ACTION ACT_LoopRead:
loopreadConditionTON(IN:=NOT setBusy AND NOT readBusy AND NOT gTBPStopLoopRead,PT:=T#1S);
IF loopreadConditionTON.Q THEN
	loopReadExcute:=TRUE;
END_IF
CASE loopReadStep OF
	0:
		IF loopReadExcute THEN
			loopReadExcute:=FALSE;
			loopReadStep:=10;
			readBusy:=TRUE;
			t1(IN:=FALSE);
			t2(IN:=FALSE);
		END_IF
	10:
		readDone:=FALSE;
		Read_State_1();
		t1(IN:=FALSE);
		loopReadStep:=loopReadStep+10;
	20:
		IF readDone THEN
			readDone:=FALSE;
			loopReadStep:=loopReadStep+10;
			t1(IN:=FALSE);
			RETURN;
		END_IF
		t1(IN:=TRUE,PT:=T#200MS);
		IF t1.Q THEN
			serialTimeOut:=TRUE;
			t1(IN:=FALSE);
			loopReadStep:=6000;
			t1(IN:=FALSE);
			RETURN;
		END_IF
	30:
		t2(IN:=TRUE,PT:=timeToNext);
		IF t2.Q THEN
			loopReadStep:=loopReadStep+10;
			t1(IN:=FALSE);
			t2(IN:=FALSE);
			RETURN;
		END_IF
	40:
		readDone:=FALSE;
		Read_State_2();
		t1(IN:=FALSE);
		loopReadStep:=loopReadStep+10;
	50:
		IF readDone THEN
			readDone:=FALSE;
			loopReadStep:=loopReadStep+10;
			t1(IN:=FALSE);
			RETURN;
		END_IF
		t1(IN:=TRUE,PT:=T#200MS);
		IF t1.Q THEN
			serialTimeOut:=TRUE;
			t1(IN:=FALSE);
			loopReadStep:=6000;
			t1(IN:=FALSE);
			RETURN;
		END_IF
	60:
		t2(IN:=TRUE,PT:=timeToNext);
		IF t2.Q THEN
			loopReadStep:=loopReadStep+10;
			t1(IN:=FALSE);
			t2(IN:=FALSE);
			RETURN;
		END_IF
	70:
		readDone:=FALSE;
		Read_State_3();
		t1(IN:=FALSE);
		loopReadStep:=loopReadStep+10;
	80:
		IF readDone THEN
			readDone:=FALSE;
			loopReadStep:=loopReadStep+10;
			t1(IN:=FALSE);
			RETURN;
		END_IF
		t1(IN:=TRUE,PT:=T#200MS);
		IF t1.Q THEN
			serialTimeOut:=TRUE;
			t1(IN:=FALSE);
			loopReadStep:=6000;
			t1(IN:=FALSE);
			RETURN;
		END_IF
	90:
		t2(IN:=TRUE,PT:=timeToNext);
		IF t2.Q THEN
			loopReadStep:=loopReadStep+10;
			t1(IN:=FALSE);
			t2(IN:=FALSE);
			RETURN;
		END_IF
	100:
		readDone:=FALSE;
		Read_State_4();
		t1(IN:=FALSE);
		loopReadStep:=loopReadStep+10;
	110:
		IF readDone THEN
			readDone:=FALSE;
			// 低位
			atTagetSpeed:=arr_RcvDataByte[6].5;
			alarm:=arr_RcvDataByte[6].3 OR arr_RcvDataByte[6].2;
			remote:=arr_RcvDataByte[6].0;
			// 高位
			acc:=arr_RcvDataByte[7].7;
			brake:=arr_RcvDataByte[7].6;
			noRotation:=arr_RcvDataByte[7].5 (*OR NOT arr_RcvDataByte[7].1*);
			loopReadStep:=loopReadStep+10;
			t1(IN:=FALSE);
			RETURN;
		END_IF
		t1(IN:=TRUE,PT:=T#200MS);
		IF t1.Q THEN
			serialTimeOut:=TRUE;
			t1(IN:=FALSE);
			loopReadStep:=6000;
			t1(IN:=FALSE);
			RETURN;
		END_IF
	120:
		t2(IN:=TRUE,PT:=timeToNext);
		IF t2.Q THEN
			t1(IN:=FALSE);
			t2(IN:=FALSE);
			loopToReadRatationTimes:=loopToReadRatationTimes+1;
			IF loopToReadRatationTimes>2 THEN // 状态读取5次，转速更新一次
				loopReadStep:=200;// 读取转速
				loopToReadRatationTimes:=0;
			ELSE
				loopReadStep:=5000;
			END_IF
			RETURN;
		END_IF
	200:
		readDone:=FALSE;
		Read_Rotation_1();
		t1(IN:=FALSE);
		loopReadStep:=loopReadStep+10;
	210:
		IF readDone THEN
			readDone:=FALSE;
			loopReadStep:=loopReadStep+10;
			t1(IN:=FALSE);
			RETURN;
		END_IF
		t1(IN:=TRUE,PT:=T#200MS);
		IF t1.Q THEN
			serialTimeOut:=TRUE;
			t1(IN:=FALSE);
			loopReadStep:=6000;
			t1(IN:=FALSE);
			RETURN;
		END_IF
	220:
		t2(IN:=TRUE,PT:=timeToNext);
		IF t2.Q THEN
			loopReadStep:=loopReadStep+10;
			t1(IN:=FALSE);
			t2(IN:=FALSE);
			RETURN;
		END_IF
	230:
		readDone:=FALSE;
		Read_Rotation_2();
		t1(IN:=FALSE);
		loopReadStep:=loopReadStep+10;
	240:
		IF readDone THEN
			readDone:=FALSE;
			loopReadStep:=loopReadStep+10;
			t1(IN:=FALSE);
			RETURN;
		END_IF
		t1(IN:=TRUE,PT:=T#200MS);
		IF t1.Q THEN
			serialTimeOut:=TRUE;
			t1(IN:=FALSE);
			loopReadStep:=6000;
			t1(IN:=FALSE);
			RETURN;
		END_IF
	250:
		t2(IN:=TRUE,PT:=timeToNext);
		IF t2.Q THEN
			loopReadStep:=loopReadStep+10;
			t1(IN:=FALSE);
			t2(IN:=FALSE);
			RETURN;
		END_IF
	260:
		readDone:=FALSE;
		Read_Rotation_3();
		t1(IN:=FALSE);
		loopReadStep:=loopReadStep+10;
	270:
		IF readDone THEN
			readDone:=FALSE;
			loopReadStep:=loopReadStep+10;
			t1(IN:=FALSE);
			RETURN;
		END_IF
		t1(IN:=TRUE,PT:=T#200MS);
		IF t1.Q THEN
			serialTimeOut:=TRUE;
			t1(IN:=FALSE);
			loopReadStep:=6000;
			RETURN;
		END_IF
	280:
		t2(IN:=TRUE,PT:=timeToNext);
		IF t2.Q THEN
			loopReadStep:=loopReadStep+10;
			t1(IN:=FALSE);
			t2(IN:=FALSE);
			RETURN;
		END_IF
	290:
		readDone:=FALSE;
		Read_Rotation_4();
		t1(IN:=FALSE);
		loopReadStep:=loopReadStep+10;
	300:
		IF readDone THEN
			readDone:=FALSE;
			intTemp:=BYTE_TO_UDINT(arr_RcvDataByte[6])*256;// 读取转速进行转换 高位
			rotationSpeed:=(intTemp+BYTE_TO_UDINT(arr_RcvDataByte[7]));// 读取转速进行转换 低位   *60  HZ 
			loopReadStep:=loopReadStep+10;
			t1(IN:=FALSE);
			RETURN;
		END_IF
		t1(IN:=TRUE,PT:=T#200MS);
		IF t1.Q THEN
			serialTimeOut:=TRUE;
			t1(IN:=FALSE);
			loopReadStep:=6000;
			t1(IN:=FALSE);
			RETURN;
		END_IF
	310:
		t2(IN:=TRUE,PT:=timeToNext);
		IF t2.Q THEN
			loopReadStep:=loopReadStep+10;
			RETURN;
		END_IF
	320:
		loopReadStep:=400;
		
	400:
		readDone:=FALSE;
		Read_TMS_1();
		t1(IN:=FALSE);
		loopReadStep:=loopReadStep+10;
	410:
		IF readDone THEN
			readDone:=FALSE;
			loopReadStep:=loopReadStep+10;
			t1(IN:=FALSE);
			RETURN;
		END_IF
		t1(IN:=TRUE,PT:=T#200MS);
		IF t1.Q THEN
			serialTimeOut:=TRUE;
			t1(IN:=FALSE);
			loopReadStep:=6000;
			RETURN;
		END_IF
	420:
		t2(IN:=TRUE,PT:=timeToNext);
		IF t2.Q THEN
			loopReadStep:=loopReadStep+10;
			t1(IN:=FALSE);
			t2(IN:=FALSE);
			RETURN;
		END_IF
	430:
		readDone:=FALSE;
		Read_TMS_2();
		t1(IN:=FALSE);
		loopReadStep:=loopReadStep+10;
	440:
		IF readDone THEN
			readDone:=FALSE;
			loopReadStep:=loopReadStep+10;
			t1(IN:=FALSE);
			RETURN;
		END_IF
		t1(IN:=TRUE,PT:=T#200MS);
		IF t1.Q THEN
			serialTimeOut:=TRUE;
			t1(IN:=FALSE);
			loopReadStep:=6000;
			RETURN;
		END_IF
	450:
		t2(IN:=TRUE,PT:=timeToNext);
		IF t2.Q THEN
			loopReadStep:=loopReadStep+10;
			t1(IN:=FALSE);
			t2(IN:=FALSE);
			RETURN;
		END_IF
	460:
		readDone:=FALSE;
		Read_TMS_3();
		t1(IN:=FALSE);
		loopReadStep:=loopReadStep+10;
	470:
		IF readDone THEN
			readDone:=FALSE;
			loopReadStep:=loopReadStep+10;
			t1(IN:=FALSE);
			RETURN;
		END_IF
		t1(IN:=TRUE,PT:=T#200MS);
		IF t1.Q THEN
			serialTimeOut:=TRUE;
			t1(IN:=FALSE);
			loopReadStep:=6000;
			RETURN;
		END_IF
	480:
		t2(IN:=TRUE,PT:=timeToNext);
		IF t2.Q THEN
			loopReadStep:=loopReadStep+10;
			t1(IN:=FALSE);
			t2(IN:=FALSE);
			RETURN;
		END_IF
	490:
		readDone:=FALSE;
		Read_TMS_4();
		t1(IN:=FALSE);
		loopReadStep:=loopReadStep+10;
	500:
		IF readDone THEN
			readDone:=FALSE;
			realTemp:=BYTE_TO_REAL(arr_RcvDataByte[6])*256;
			tMSTemperature:=(realTemp+BYTE_TO_REAL(arr_RcvDataByte[7]))/10;
			loopReadStep:=loopReadStep+10;
			t1(IN:=FALSE);
			RETURN;
		END_IF
		t1(IN:=TRUE,PT:=T#200MS);
		IF t1.Q THEN
			serialTimeOut:=TRUE;
			t1(IN:=FALSE);
			loopReadStep:=6000;
			RETURN;
		END_IF
	510:
		t2(IN:=TRUE,PT:=timeToNext);
		IF t2.Q THEN
			loopReadStep:=loopReadStep+10;
			RETURN;
		END_IF
	520:
		loopReadStep:=5000;
	5000:
		loopReadStep:=0;
		readBusy:=FALSE;
		readDone:=FALSE;
		serialTimeOutTimes:=0;
	6000:
		timeoutResetTime(IN:=TRUE,PT:=T#0.5S);
		IF timeoutResetTime.Q THEN
			readDone:=FALSE;
			loopReadStep:=0;
			readBusy:=FALSE;
			timeoutResetTime(IN:=FALSE);
			serialTimeOutTimes:=serialTimeOutTimes+1;
			IF serialTimeOutTimes>5 THEN
				serialTimeOutTimes:=0;
				serialTimeoutError:=TRUE;
			END_IF
		END_IF
END_CASE
END_ACTION

ACTION ACT_Reset:

CASE resetStep OF
	0:
	IF resetExcute THEN
		IF NOT resetBusy THEN
			resetExcute:=FALSE;
			resetBusy:=FALSE;
			resetDone:=FALSE;
			resetError:=FALSE;
			stopBusy:=FALSE;
			stopDone:=FALSE;
			stopError:=FALSE;
			startBusy:=FALSE;
			startDone:=FALSE;
			startError:=FALSE;
			serialError:=FALSE;
			serialDone:=FALSE;
			serialError:=FALSE;
			serialTimeOut:=FALSE;
			serialRecError:=FALSE;
			serialStep:=0;
			startStep:=0;
			stopStep:=0;
			resetStep:=90;
		END_IF
	END_IF
	Timerreset(IN:= FALSE);
	TimerresetTOut(IN:= FALSE);
	;
	
	90:
		IF loopReadStep<10 AND startStep<10 AND stopStep<10 THEN
			readDone:=FALSE;
			Set_Reset_1();
			resetStep:=100;
		END_IF
	100:
		IF readDone THEN
			readDone:=FALSE;
			resetStep:=resetStep+10;
			TimerresetTOut(IN:=FALSE);
			RETURN;
		END_IF
		TimerresetTOut(IN:=TRUE,PT:=T#200MS);
		IF TimerresetTOut.Q THEN
			serialTimeOut:=TRUE;
			TimerresetTOut(IN:=FALSE);
			resetStep:=6000;
			RETURN;
		END_IF
	110:
		Timerreset(IN:= NOT Timerreset.q, PT:=T#30MS);
		IF Timerreset.Q THEN
			resetStep:=resetStep+10;
			Timerreset(IN:= FALSE);
		END_IF
	120:
		readDone:=FALSE;
		Set_Reset_2();
		resetStep:=resetStep+10;
	130:
		IF readDone THEN
			readDone:=FALSE;
			resetStep:=resetStep+10;
			TimerresetTOut(IN:=FALSE);
			RETURN;
		END_IF
		TimerresetTOut(IN:=TRUE,PT:=T#200MS);
		IF TimerresetTOut.Q THEN
			serialTimeOut:=TRUE;
			TimerresetTOut(IN:=FALSE);
			resetStep:=6000;
			RETURN;
		END_IF
	140:
		Timerreset(IN:= NOT Timerreset.q, PT:=T#30MS);
		IF Timerreset.Q THEN
			resetStep:=resetStep+10;
			Timerreset(IN:= FALSE);
		END_IF
	150:
		readDone:=FALSE;
		Set_Reset_3();
		resetStep:=resetStep+10;
	160:
		IF readDone THEN
			readDone:=FALSE;
			resetStep:=resetStep+10;
			TimerresetTOut(IN:=FALSE);
			RETURN;
		END_IF
		TimerresetTOut(IN:=TRUE,PT:=T#200MS);
		IF TimerresetTOut.Q THEN
			serialTimeOut:=TRUE;
			TimerresetTOut(IN:=FALSE);
			resetStep:=6000;
			RETURN;
		END_IF
	170:
		Timerreset(IN:= NOT Timerreset.q, PT:=T#30MS);
		IF Timerreset.Q THEN
			resetStep:=resetStep+10;
			Timerreset(IN:= FALSE);
		END_IF
	180:
		readDone:=FALSE;
		Set_Reset_4();
		resetStep:=resetStep+10;
	190:
		IF readDone THEN
			readDone:=FALSE;
			resetStep:=resetStep+10;
			TimerresetTOut(IN:=FALSE);
			RETURN;
		END_IF
		TimerresetTOut(IN:=TRUE,PT:=T#200MS);
		IF TimerresetTOut.Q THEN
			serialTimeOut:=TRUE;
			TimerresetTOut(IN:=FALSE);
			resetStep:=6000;
			RETURN;
		END_IF
	200:
		Timerreset(IN:= NOT Timerreset.q, PT:=T#10MS);
		IF Timerreset.Q THEN
			resetStep:=resetStep+10;
			Timerreset(IN:= FALSE);
		END_IF
	210:
		resetStep:=5000;
	;
	5000://done
		resetBusy:=FALSE;
		resetDone:=TRUE;
		resetError:=FALSE;
		resetStep:=0;
		readDone:=FALSE;
	;
	6000://error
		resetBusy:=FALSE;
		resetDone:=FALSE;
		resetError:=TRUE;
		resetStep:=0;
		readDone:=FALSE;
	;
	
END_CASE
END_ACTION

ACTION ACT_Send:

CASE serialStep OF
	0:
	IF serialExcute THEN
		serialExcute:=FALSE;
		IF NOT serialBusy THEN
			serialStep:=90;
			serialBusy:=TRUE;
			serialDone:=FALSE;
			serialError:=FALSE;
			serialTimeOut:=FALSE;
			serialRecError:=FALSE;
			serialTimeOut:=FALSE;
		END_IF
	END_IF
	Timer1(IN:= FALSE);
	;
	
	90:
		arr_SendData:=sendbyte;
		serialStep:=100;
	100:
		send1(
			pSendData:= ADR(arr_SendData), 
			Length:= sendLenght, 
			Busy=> , 
			Error=> , 
			TXbuffer:= gTxBuffer_TBP);
		serialStep:=serialStep+10;
	110:
		Timer1(IN:= NOT timer1.q, PT:=T#10MS);
		IF Timer1.Q THEN
			serialStep:=serialStep+10;
			Timer1(IN:= FALSE);
		END_IF
	120:
		Timer1(IN:= NOT timer1.q, PT:=T#500MS);
		IF Timer1.Q THEN
			serialStep:=6000;
			Timer1(IN:= FALSE);
			serialTimeOut:=TRUE;
			RETURN;
		END_IF
		IF NOT send1.busy  THEN
			Timer1(IN:= FALSE);
			serialTimeOut:=FALSE;
			serialStep:=200;
		END_IF
		IF send1.Error <> COMERROR_NOERROR THEN
			serialRecError:=TRUE;
		END_IF
	200://数据处理
		serialStep:=serialStep+10;
	210:
		Timer1(IN:= NOT timer1.q, PT:=T#10MS);
		IF Timer1.Q THEN
			serialStep:=serialStep+10;
			Timer1(IN:= FALSE);
		END_IF
	220:
		//数据转换
		Timer1(IN:= FALSE);
		serialStep:=1000;
	
	1000:
		Timer1(IN:= NOT timer1.q, PT:=T#50MS);
		IF Timer1.Q THEN
			serialStep:=5000;
			Timer1(IN:= FALSE);
			// sendstr:='';
			serialTimeOut:=FALSE;
		END_IF
	;
	5000://done
		serialBusy:=FALSE;
		serialDone:=TRUE;
		serialError:=FALSE;
		serialStep:=0;
	;
	6000://error
		serialBusy:=FALSE;
		serialDone:=FALSE;
		serialError:=TRUE;
		serialStep:=0;
	;
	
END_CASE
END_ACTION

ACTION ACT_Start:

CASE startStep OF
	0:
	IF startExcute THEN
		IF NOT startBusy THEN
			startExcute:=FALSE;
			startBusy:=FALSE;
			startDone:=FALSE;
			startError:=FALSE;
			startStep:=90;
			serialTimeOut:=FALSE;
			gTBPStopLoopRead:=true;
		END_IF
	END_IF
	TimerStart(IN:= FALSE);
	TimerStartTOut(IN:= FALSE);
	;
	
	90:
		IF loopReadStep<10 AND resetStep<10 AND stopStep<10 THEN
			readDone:=FALSE;
			Set_Start_0();
			startStep:=100;
		END_IF
	100:
		IF readDone THEN
			readDone:=FALSE;
			startStep:=startStep+10;
			TimerStartTOut(IN:=FALSE);
			RETURN;
		END_IF
		TimerStartTOut(IN:=TRUE,PT:=T#2000MS);
		IF TimerStartTOut.Q THEN
			serialTimeOut:=TRUE;
			TimerStartTOut(IN:=FALSE);
			startStep:=6000;
			RETURN;
		END_IF
	110:
		TimerStart(IN:= NOT TimerStart.q, PT:=T#30MS);
		IF TimerStart.Q THEN
			startStep:=startStep+10;
			TimerStart(IN:= FALSE);
		END_IF
	120:
		readDone:=FALSE;
		Set_Start_Stop_1();
		startStep:=startStep+10;
	130:
		IF readDone THEN
			readDone:=FALSE;
			startStep:=startStep+10;
			TimerStartTOut(IN:=FALSE);
			RETURN;
		END_IF
		TimerStartTOut(IN:=TRUE,PT:=T#2000MS);
		IF TimerStartTOut.Q THEN
			serialTimeOut:=TRUE;
			TimerStartTOut(IN:=FALSE);
			startStep:=6000;
			RETURN;
		END_IF
	140:
		TimerStart(IN:= NOT TimerStart.q, PT:=T#30MS);
		IF TimerStart.Q THEN
			startStep:=startStep+10;
			TimerStart(IN:= FALSE);
		END_IF
	150:
		readDone:=FALSE;
		Set_Start_Stop_2();
		startStep:=startStep+10;
	160:
		IF readDone THEN
			readDone:=FALSE;
			startStep:=startStep+10;
			TimerStartTOut(IN:=FALSE);
			RETURN;
		END_IF
		TimerStartTOut(IN:=TRUE,PT:=T#2000MS);
		IF TimerStartTOut.Q THEN
			serialTimeOut:=TRUE;
			TimerStartTOut(IN:=FALSE);
			startStep:=6000;
			RETURN;
		END_IF
	170:
		TimerStart(IN:= NOT TimerStart.q, PT:=T#30MS);
		IF TimerStart.Q THEN
			startStep:=startStep+10;
			TimerStart(IN:= FALSE);
		END_IF
	180:
		readDone:=FALSE;
		Set_Start_Stop_3();
		startStep:=startStep+10;
	190:
		IF readDone THEN
			readDone:=FALSE;
			startStep:=startStep+10;
			TimerStartTOut(IN:=FALSE);
			RETURN;
		END_IF
		TimerStartTOut(IN:=TRUE,PT:=T#2000MS);
		IF TimerStartTOut.Q THEN
			serialTimeOut:=TRUE;
			TimerStartTOut(IN:=FALSE);
			startStep:=6000;
			RETURN;
		END_IF
	200:
		TimerStart(IN:= NOT TimerStart.q, PT:=T#30MS);
		IF TimerStart.Q THEN
			startStep:=startStep+10;
			TimerStart(IN:= FALSE);
		END_IF
	210:
		startStep:=5000;
	;
	5000://done
		startBusy:=FALSE;
		startDone:=TRUE;
		startError:=FALSE;
		startStep:=0;
		readDone:=FALSE;
	;
	6000://error
		startBusy:=FALSE;
		startDone:=FALSE;
		startError:=TRUE;
		startStep:=0;
		readDone:=FALSE;
	;
	
END_CASE
END_ACTION

ACTION ACT_Stop:

CASE stopStep OF
	0:
	IF stopExcute THEN
		IF NOT stopBusy THEN
			stopExcute:=FALSE;
			stopBusy:=FALSE;
			stopDone:=FALSE;
			stopError:=FALSE;
			stopStep:=90;
			serialTimeOut:=FALSE;
			gTBPStopLoopRead:=TRUE;
		END_IF
	END_IF
	Timerstop(IN:= FALSE);
	TimerstopTOut(IN:= FALSE);
	;
	
	90:
		IF loopReadStep<10 AND resetStep<10 AND startStep<10 THEN
			readDone:=FALSE;
			Set_stop_0();
			stopStep:=100;
		END_IF
	100:
		IF readDone THEN
			readDone:=FALSE;
			stopStep:=stopStep+10;
			TimerstopTOut(IN:=FALSE);
			RETURN;
		END_IF
		TimerstopTOut(IN:=TRUE,PT:=T#200MS);
		IF TimerstopTOut.Q THEN
			serialTimeOut:=TRUE;
			TimerstopTOut(IN:=FALSE);
			stopStep:=6000;
			RETURN;
		END_IF
	110:
		Timerstop(IN:= NOT Timerstop.q, PT:=T#30MS);
		IF Timerstop.Q THEN
			stopStep:=stopStep+10;
			Timerstop(IN:= FALSE);
		END_IF
	120:
		readDone:=FALSE;
		Set_Start_Stop_1();
		stopStep:=stopStep+10;
	130:
		IF readDone THEN
			readDone:=FALSE;
			stopStep:=stopStep+10;
			TimerstopTOut(IN:=FALSE);
			RETURN;
		END_IF
		TimerstopTOut(IN:=TRUE,PT:=T#200MS);
		IF TimerstopTOut.Q THEN
			serialTimeOut:=TRUE;
			TimerstopTOut(IN:=FALSE);
			stopStep:=6000;
			RETURN;
		END_IF
	140:
		Timerstop(IN:= NOT Timerstop.q, PT:=T#30MS);
		IF Timerstop.Q THEN
			stopStep:=stopStep+10;
			Timerstop(IN:= FALSE);
		END_IF
	150:
		readDone:=FALSE;
		Set_Start_Stop_2();
		stopStep:=stopStep+10;
	160:
		IF readDone THEN
			readDone:=FALSE;
			stopStep:=stopStep+10;
			TimerstopTOut(IN:=FALSE);
			RETURN;
		END_IF
		TimerstopTOut(IN:=TRUE,PT:=T#200MS);
		IF TimerstopTOut.Q THEN
			serialTimeOut:=TRUE;
			TimerstopTOut(IN:=FALSE);
			stopStep:=6000;
			RETURN;
		END_IF
	170:
		Timerstop(IN:= NOT Timerstop.q, PT:=T#30MS);
		IF Timerstop.Q THEN
			stopStep:=stopStep+10;
			Timerstop(IN:= FALSE);
		END_IF
	180:
		readDone:=FALSE;
		Set_Start_Stop_3();
		stopStep:=stopStep+10;
	190:
		IF readDone THEN
			readDone:=FALSE;
			stopStep:=stopStep+10;
			TimerstopTOut(IN:=FALSE);
			RETURN;
		END_IF
		TimerstopTOut(IN:=TRUE,PT:=T#200MS);
		IF TimerstopTOut.Q THEN
			serialTimeOut:=TRUE;
			TimerstopTOut(IN:=FALSE);
			stopStep:=6000;
			RETURN;
		END_IF
	200:
		Timerstop(IN:= NOT Timerstop.q, PT:=T#30MS);
		IF Timerstop.Q THEN
			stopStep:=stopStep+10;
			Timerstop(IN:= FALSE);
		END_IF
	210:
		stopStep:=5000;
	;
	5000://done
		stopBusy:=FALSE;
		stopDone:=TRUE;
		stopError:=FALSE;
		stopStep:=0;
		readDone:=FALSE;
		gTBPStopLoopRead:=FALSE;
	;
	6000://error
		stopBusy:=FALSE;
		stopDone:=FALSE;
		stopError:=TRUE;
		stopStep:=0;
		readDone:=FALSE;
		gTBPStopLoopRead:=FALSE;
	;
	
END_CASE
END_ACTION

METHOD CalASII_Byte : UDINT
VAR_INPUT
	date1:UDINT;
END_VAR
IF date1=10 THEN
	CalASII_Byte:=41;
END_IF
IF date1=11 THEN
	CalASII_Byte:=42;
END_IF
IF date1=12 THEN
	CalASII_Byte:=43;
END_IF
IF date1=13 THEN
	CalASII_Byte:=44;
END_IF
IF date1=14 THEN
	CalASII_Byte:=45;
END_IF
IF date1=15 THEN
	CalASII_Byte:=46;
END_IF
IF date1<10 THEN
	CalASII_Byte:=date1+30;
END_IF
IF date1>15 THEN
	CalASII_Byte:=date1+30;
END_IF
END_METHOD

METHOD Interface_Reset : BOOL
VAR_INPUT

END_VAR
VAR

END_VAR
resetExcute:=true;
END_METHOD

METHOD Interface_Start : BOOL
VAR_INPUT

END_VAR
VAR
END_VAR
startExcute:=true;
END_METHOD

METHOD Interface_Stop : BOOL
VAR_INPUT

END_VAR
VAR

END_VAR
stopExcute:=true;
END_METHOD

METHOD Read_Rotation_1 : BOOL
VAR_INPUT

END_VAR
VAR
	sumq:UDINT;
	mod128:UDINT;
	intTemp:INT;
END_VAR
sendLenght:=15;
sendbyte[1]:=16#02;
sendbyte[2]:=16#01;
sendbyte[3]:=16#00;
sendbyte[4]:=16#0A;
sendbyte[5]:=16#57;
sendbyte[6]:=16#00;
sendbyte[7]:=16#02;
sendbyte[8]:=16#80;
sendbyte[9]:=16#80;
sendbyte[10]:=16#9A;
sendbyte[11]:=16#00;
sendbyte[12]:=16#01;
sendbyte[13]:=16#FF;
sendbyte[14]:=16#03;
sendbyte[15]:=16#03;
serialExcute:=TRUE;
END_METHOD

METHOD Read_Rotation_2 : BOOL
VAR_INPUT

END_VAR
VAR
	sumq:UDINT;
	mod128:UDINT;
	intTemp:INT;
END_VAR
sendLenght:=15;
sendbyte[1]:=16#02;
sendbyte[2]:=16#01;
sendbyte[3]:=16#00;
sendbyte[4]:=16#0A;
sendbyte[5]:=16#57;
sendbyte[6]:=16#00;
sendbyte[7]:=16#02;
sendbyte[8]:=16#80;
sendbyte[9]:=16#81;
sendbyte[10]:=16#99;
sendbyte[11]:=16#00;
sendbyte[12]:=16#55;
sendbyte[13]:=16#AB;
sendbyte[14]:=16#03;
sendbyte[15]:=16#03;
serialExcute:=TRUE;
END_METHOD

METHOD Read_Rotation_3 : BOOL
VAR_INPUT

END_VAR
VAR
	sumq:UDINT;
	mod128:UDINT;
	intTemp:INT;
END_VAR
sendLenght:=14;
sendbyte[1]:=16#02;
sendbyte[2]:=16#01;
sendbyte[3]:=16#00;
sendbyte[4]:=16#09;
sendbyte[5]:=16#52;
sendbyte[6]:=16#00;
sendbyte[7]:=16#02;
sendbyte[8]:=16#80;
sendbyte[9]:=16#81;
sendbyte[10]:=16#00;
sendbyte[11]:=16#02;
sendbyte[12]:=16#9D;
sendbyte[13]:=16#03;
sendbyte[14]:=16#03;
serialExcute:=TRUE;
END_METHOD

METHOD Read_Rotation_4 : BOOL
VAR_INPUT

END_VAR
VAR
	sumq:UDINT;
	mod128:UDINT;
	intTemp:INT;
END_VAR
sendLenght:=14;
sendbyte[1]:=16#02;
sendbyte[2]:=16#01;
sendbyte[3]:=16#00;
sendbyte[4]:=16#09;
sendbyte[5]:=16#52;
sendbyte[6]:=16#00;
sendbyte[7]:=16#02;
sendbyte[8]:=16#80;
sendbyte[9]:=16#82;
sendbyte[10]:=16#00;
sendbyte[11]:=16#02;
sendbyte[12]:=16#9C;
sendbyte[13]:=16#03;
sendbyte[14]:=16#03;
serialExcute:=TRUE;
END_METHOD

METHOD Read_State_1 : BOOL
VAR_INPUT

END_VAR
VAR
	sumq:UDINT;
	mod128:UDINT;
	intTemp:INT;
END_VAR
sendLenght:=15;
sendbyte[1]:=16#02;
sendbyte[2]:=16#01;
sendbyte[3]:=16#00;
sendbyte[4]:=16#0A;
sendbyte[5]:=16#57;
sendbyte[6]:=16#00;
sendbyte[7]:=16#02;
sendbyte[8]:=16#80;
sendbyte[9]:=16#80;
sendbyte[10]:=16#9A;
sendbyte[11]:=16#00;
sendbyte[12]:=16#40;
sendbyte[13]:=16#C0;
sendbyte[14]:=16#03;
sendbyte[15]:=16#03;
serialExcute:=TRUE;
END_METHOD

METHOD Read_State_2 : BOOL
VAR_INPUT

END_VAR
VAR
	sumq:UDINT;
	mod128:UDINT;
	intTemp:INT;
END_VAR
sendLenght:=15;
sendbyte[1]:=16#02;
sendbyte[2]:=16#01;
sendbyte[3]:=16#00;
sendbyte[4]:=16#0A;
sendbyte[5]:=16#57;
sendbyte[6]:=16#00;
sendbyte[7]:=16#02;
sendbyte[8]:=16#80;
sendbyte[9]:=16#81;
sendbyte[10]:=16#99;
sendbyte[11]:=16#00;
sendbyte[12]:=16#55;
sendbyte[13]:=16#AB;
sendbyte[14]:=16#03;
sendbyte[15]:=16#03;
serialExcute:=TRUE;
END_METHOD

METHOD Read_State_3 : BOOL
VAR_INPUT

END_VAR
VAR
	sumq:UDINT;
	mod128:UDINT;
	intTemp:INT;
END_VAR
sendLenght:=14;
sendbyte[1]:=16#02;
sendbyte[2]:=16#01;
sendbyte[3]:=16#00;
sendbyte[4]:=16#09;
sendbyte[5]:=16#52;
sendbyte[6]:=16#00;
sendbyte[7]:=16#02;
sendbyte[8]:=16#80;
sendbyte[9]:=16#81;
sendbyte[10]:=16#00;
sendbyte[11]:=16#02;
sendbyte[12]:=16#9D;
sendbyte[13]:=16#03;
sendbyte[14]:=16#03;
serialExcute:=TRUE;
END_METHOD

METHOD Read_State_4 : BOOL
VAR_INPUT

END_VAR
VAR
	sumq:UDINT;
	mod128:UDINT;
	intTemp:INT;
END_VAR
sendLenght:=14;
sendbyte[1]:=16#02;
sendbyte[2]:=16#01;
sendbyte[3]:=16#00;
sendbyte[4]:=16#09;
sendbyte[5]:=16#52;
sendbyte[6]:=16#00;
sendbyte[7]:=16#02;
sendbyte[8]:=16#80;
sendbyte[9]:=16#82;
sendbyte[10]:=16#00;
sendbyte[11]:=16#02;
sendbyte[12]:=16#9C;
sendbyte[13]:=16#03;
sendbyte[14]:=16#03;
serialExcute:=TRUE;
END_METHOD

METHOD Read_TMS_1 : BOOL
VAR_INPUT

END_VAR
VAR
	sumq:UDINT;
	mod128:UDINT;
	intTemp:INT;
END_VAR
sendLenght:=15;
sendbyte[1]:=16#02;
sendbyte[2]:=16#01;
sendbyte[3]:=16#00;
sendbyte[4]:=16#0A;
sendbyte[5]:=16#57;
sendbyte[6]:=16#00;
sendbyte[7]:=16#02;
sendbyte[8]:=16#80;
sendbyte[9]:=16#80;
sendbyte[10]:=16#9A;
sendbyte[11]:=16#00;
sendbyte[12]:=16#11;
sendbyte[13]:=16#EF;
sendbyte[14]:=16#03;
sendbyte[15]:=16#03;
serialExcute:=TRUE;
END_METHOD

METHOD Read_TMS_2 : BOOL
VAR_INPUT

END_VAR
VAR
	sumq:UDINT;
	mod128:UDINT;
	intTemp:INT;
END_VAR
sendLenght:=15;
sendbyte[1]:=16#02;
sendbyte[2]:=16#01;
sendbyte[3]:=16#00;
sendbyte[4]:=16#0A;
sendbyte[5]:=16#57;
sendbyte[6]:=16#00;
sendbyte[7]:=16#02;
sendbyte[8]:=16#80;
sendbyte[9]:=16#81;
sendbyte[10]:=16#99;
sendbyte[11]:=16#00;
sendbyte[12]:=16#55;
sendbyte[13]:=16#AB;
sendbyte[14]:=16#03;
sendbyte[15]:=16#03;
serialExcute:=TRUE;
END_METHOD

METHOD Read_TMS_3 : BOOL
VAR_INPUT

END_VAR
VAR
	sumq:UDINT;
	mod128:UDINT;
	intTemp:INT;
END_VAR
sendLenght:=14;
sendbyte[1]:=16#02;
sendbyte[2]:=16#01;
sendbyte[3]:=16#00;
sendbyte[4]:=16#09;
sendbyte[5]:=16#52;
sendbyte[6]:=16#00;
sendbyte[7]:=16#02;
sendbyte[8]:=16#80;
sendbyte[9]:=16#81;
sendbyte[10]:=16#00;
sendbyte[11]:=16#02;
sendbyte[12]:=16#9D;
sendbyte[13]:=16#03;
sendbyte[14]:=16#03;
serialExcute:=TRUE;
END_METHOD

METHOD Read_TMS_4 : BOOL
VAR_INPUT

END_VAR
VAR
	sumq:UDINT;
	mod128:UDINT;
	intTemp:INT;
END_VAR
sendLenght:=14;
sendbyte[1]:=16#02;
sendbyte[2]:=16#01;
sendbyte[3]:=16#00;
sendbyte[4]:=16#09;
sendbyte[5]:=16#52;
sendbyte[6]:=16#00;
sendbyte[7]:=16#02;
sendbyte[8]:=16#80;
sendbyte[9]:=16#82;
sendbyte[10]:=16#00;
sendbyte[11]:=16#02;
sendbyte[12]:=16#9C;
sendbyte[13]:=16#03;
sendbyte[14]:=16#03;
serialExcute:=TRUE;
END_METHOD

METHOD Set_Reset_1 : BOOL
VAR
	sumq:UDINT;
	mod128:UDINT;
	intTemp:INT;
END_VAR
sendLenght:=15;
sendbyte[1]:=16#02;
sendbyte[2]:=16#01;
sendbyte[3]:=16#00;
sendbyte[4]:=16#0A;
sendbyte[5]:=16#57;
sendbyte[6]:=16#00;
sendbyte[7]:=16#02;
sendbyte[8]:=16#80;
sendbyte[9]:=16#80;
sendbyte[10]:=16#9A;
sendbyte[11]:=16#00;
sendbyte[12]:=16#41;
sendbyte[13]:=16#BF;
sendbyte[14]:=16#03;
sendbyte[15]:=16#03;
serialExcute:=TRUE;
END_METHOD

METHOD Set_Reset_2 : BOOL
VAR
	sumq:UDINT;
	mod128:UDINT;
	intTemp:INT;
END_VAR
sendLenght:=15;
sendbyte[1]:=16#02;
sendbyte[2]:=16#01;
sendbyte[3]:=16#00;
sendbyte[4]:=16#0A;
sendbyte[5]:=16#57;
sendbyte[6]:=16#00;
sendbyte[7]:=16#02;
sendbyte[8]:=16#80;
sendbyte[9]:=16#82;
sendbyte[10]:=16#98;
sendbyte[11]:=16#00;
sendbyte[12]:=16#44;
sendbyte[13]:=16#BC;
sendbyte[14]:=16#03;
sendbyte[15]:=16#03;
serialExcute:=TRUE;
END_METHOD

METHOD Set_Reset_3 : BOOL

VAR
	sumq:UDINT;
	mod128:UDINT;
	intTemp:INT;
END_VAR
sendLenght:=15;
sendbyte[1]:=16#02;
sendbyte[2]:=16#01;
sendbyte[3]:=16#00;
sendbyte[4]:=16#0A;
sendbyte[5]:=16#57;
sendbyte[6]:=16#00;
sendbyte[7]:=16#02;
sendbyte[8]:=16#80;
sendbyte[9]:=16#81;
sendbyte[10]:=16#99;
sendbyte[11]:=16#00;
sendbyte[12]:=16#AA;
sendbyte[13]:=16#56;
sendbyte[14]:=16#03;
sendbyte[15]:=16#03;
serialExcute:=TRUE;
END_METHOD

METHOD Set_Reset_4 : BOOL

VAR
	sumq:UDINT;
	mod128:UDINT;
	intTemp:INT;
END_VAR
sendLenght:=14;
sendbyte[1]:=16#02;
sendbyte[2]:=16#01;
sendbyte[3]:=16#00;
sendbyte[4]:=16#09;
sendbyte[5]:=16#52;
sendbyte[6]:=16#00;
sendbyte[7]:=16#02;
sendbyte[8]:=16#80;
sendbyte[9]:=16#81;
sendbyte[10]:=16#00;
sendbyte[11]:=16#02;
sendbyte[12]:=16#9D;
sendbyte[13]:=16#03;
sendbyte[14]:=16#03;
serialExcute:=TRUE;
END_METHOD

METHOD Set_Start_0 : BOOL
VAR
	sumq:UDINT;
	mod128:UDINT;
	intTemp:INT;
END_VAR
sendLenght:=15;
sendbyte[1]:=16#02;
sendbyte[2]:=16#01;
sendbyte[3]:=16#00;
sendbyte[4]:=16#0A;
sendbyte[5]:=16#57;
sendbyte[6]:=16#00;
sendbyte[7]:=16#02;
sendbyte[8]:=16#80;
sendbyte[9]:=16#80;
sendbyte[10]:=16#9A;
sendbyte[11]:=16#00;
sendbyte[12]:=16#08;
sendbyte[13]:=16#F8;
sendbyte[14]:=16#03;
sendbyte[15]:=16#03;
serialExcute:=TRUE;
END_METHOD

METHOD Set_Start_Stop_1 : BOOL
VAR
	sumq:UDINT;
	mod128:UDINT;
	intTemp:INT;
END_VAR
sendLenght:=15;
sendbyte[1]:=16#02;
sendbyte[2]:=16#01;
sendbyte[3]:=16#00;
sendbyte[4]:=16#0A;
sendbyte[5]:=16#57;
sendbyte[6]:=16#00;
sendbyte[7]:=16#02;
sendbyte[8]:=16#80;
sendbyte[9]:=16#82;
sendbyte[10]:=16#98;
sendbyte[11]:=16#00;
sendbyte[12]:=16#01;
sendbyte[13]:=16#FF;
sendbyte[14]:=16#03;
sendbyte[15]:=16#03;
serialExcute:=TRUE;
END_METHOD

METHOD Set_Start_Stop_2 : BOOL

VAR
	sumq:UDINT;
	mod128:UDINT;
	intTemp:INT;
END_VAR
sendLenght:=15;
sendbyte[1]:=16#02;
sendbyte[2]:=16#01;
sendbyte[3]:=16#00;
sendbyte[4]:=16#0A;
sendbyte[5]:=16#57;
sendbyte[6]:=16#00;
sendbyte[7]:=16#02;
sendbyte[8]:=16#80;
sendbyte[9]:=16#81;
sendbyte[10]:=16#99;
sendbyte[11]:=16#00;
sendbyte[12]:=16#AA;
sendbyte[13]:=16#56;
sendbyte[14]:=16#03;
sendbyte[15]:=16#03;
serialExcute:=TRUE;
END_METHOD

METHOD Set_Start_Stop_3 : BOOL

VAR
	sumq:UDINT;
	mod128:UDINT;
	intTemp:INT;
END_VAR
sendLenght:=14;
sendbyte[1]:=16#02;
sendbyte[2]:=16#01;
sendbyte[3]:=16#00;
sendbyte[4]:=16#09;
sendbyte[5]:=16#52;
sendbyte[6]:=16#00;
sendbyte[7]:=16#02;
sendbyte[8]:=16#80;
sendbyte[9]:=16#81;
sendbyte[10]:=16#00;
sendbyte[11]:=16#02;
sendbyte[12]:=16#9D;
sendbyte[13]:=16#03;
sendbyte[14]:=16#03;
serialExcute:=TRUE;
END_METHOD

METHOD Set_Stop_0 : BOOL

VAR
	sumq:UDINT;
	mod128:UDINT;
	intTemp:INT;
END_VAR
sendLenght:=15;
sendbyte[1]:=16#02;
sendbyte[2]:=16#01;
sendbyte[3]:=16#00;
sendbyte[4]:=16#0A;
sendbyte[5]:=16#57;
sendbyte[6]:=16#00;
sendbyte[7]:=16#02;
sendbyte[8]:=16#80;
sendbyte[9]:=16#80;
sendbyte[10]:=16#9A;
sendbyte[11]:=16#00;
sendbyte[12]:=16#09;
sendbyte[13]:=16#F7;
sendbyte[14]:=16#03;
sendbyte[15]:=16#03;
serialExcute:=TRUE;
END_METHOD

END_PROGRAM

// ---- POUs/BaseModule/ActionModule/VPEModule/VPEModule.TcPOU
(*
--报错编号0: 无报错
--报错编号1: openend Error
--报错编号2: closeract Error
*)
FUNCTION_BLOCK VPEModule
VAR_IN_OUT
	WarmHMI					:WARMStruct;
	NoteHMI					:NoteStruct;
	operatorLog				:printLogModule_EX;
END_VAR
VAR_INPUT
	VPEType						:VPEType:=VPEType_Default;//设置泵组的类型
	real_TimeMonitor			:BOOL:=TRUE;//实时状态检测
	enabletcp					:BOOL:=TRUE;//启用TCP读取参数
	tcpSendDelayTime			:TIME:=T#0.5S;
	ACCMaxtime					:TIME:=T#30S;
	DCCMaxtime					:TIME:=T#10S;
	open						:BOOL:=FALSE;//启动触发信号
	openCondition				:BOOL:=TRUE;//启动条件
	close						:BOOL:=FALSE;//停止触发信号
	closeCondition				:BOOL:=TRUE;//停止条件
	reset						:BOOL:=FALSE;//复位信号
	stop						:BOOL:=FALSE;//停止信号
	power						:BOOL:=TRUE;//泵组动作后是否关闭继电器得电状态, TRUE--保持得电,FALSE--断开得电
	enable						:BOOL:=TRUE;//泵组禁用条件
	//ctrlMode					:ControlMode:=ControlMode.eManualCtrMode;//eManualCtrMode or eAutoCtrMode
	hmiEN						:BOOL:=TRUE;//HMI 启用条件
	
	errorDelayTime				:TIME:=T#5000MS;//泵组感应器感应超时		
	
	doneDelayTimeShortopenend	:TIME:=T#100MS;//泵组启动感应到位延时_伸出
	doneDelayTimeShortcloseract	:TIME:=T#50MS;//泵组感应到位延时_收回
	doneDelayTimeLongopenend	:TIME:=T#500MS;//无泵组感应到位延时_伸出
	doneDelayTimeLongcloseract	:TIME:=T#50MS;//无泵组感应到位延时_收回
	errorID						:UDINT:=0;//泵组错误报警分配的起始ID
	nameTXT						:STRING(255):='';//泵组名字
	
	Accing						:BOOL;// 加速中
	Dccing						:BOOL;// 减速中
	Normal						:BOOL;// 泵组全速中

	AccAprSw					:BOOL:=FALSE;// 泵组预热加速启动信号,需要链接到实际的IO点
	AlmAprSw					:BOOL:=FALSE;// 泵组报警信号,需要链接到实际的IO点;有信号，无报错
	
	sHost						:STRING(20):='127.0.0.1';// 通讯IP地址; server时表示本地host; client时表示远程host
	nPort						:UDINT:=8900;// 通讯端口号;
	bEnable						:BOOL:=TRUE;// 通讯启用\禁用连接
	sSendSuffix					:STRING:='';//此处可统一添加发送后缀字符 $R$N
	slaveID						:UINT;// 从站号
	noteWTXT_open				:WSTRING(255):="";// 泵组打开动作NoteTXT 中文
	noteWTXT_close				:WSTRING(255):="";// 泵组关闭动作NoteTXT 中文
END_VAR
VAR_OUTPUT
	note_open				:BOOL:=FALSE;// 开执行条件不满足提示
	note_close				:BOOL:=FALSE;// 关执行条件不满足提示
	openRelay				:BOOL:=FALSE;// 泵组启动执行继电器,需要链接到实际的IO点
	closeRelay				:BOOL:=FALSE;// 泵组停止执行继电器,需要链接到实际的IO点
	resetRelay				:BOOL:=FALSE;// 泵组复位执行继电器,需要链接到实际的IO点
	
	bDryPump				:BOOL;// 螺杆泵启动状态
	bBooster				:BOOL;// 罗茨泵启动状态
	VPEStart				:BOOL;// 泵组运行状态
	runTime						: LINT;// 泵组运行时间
	DryPumpSpeed			:DWORD:=0;// 螺杆泵速度
	DryPumpTemperature		:DWORD:=0;// 螺杆泵温度
	DryPumpCurrent			:DWORD:=0;// 螺杆泵电流
	DryPumpPower			:DWORD:=0;// 螺杆泵功率
	
	DryPumpAlm				:BOOL;// 螺杆泵报警标志位
	
	BoosterSpeed			:DWORD:=0;// 罗茨泵速度
	BoosterTemperature		:DWORD:=0;// 罗茨泵温度
	BoosterCurrent			:DWORD:=0;// 罗茨泵电流
	BoosterPower			:DWORD:=0;// 罗茨泵功率
	
	BoosterAlm				:BOOL;// 罗茨泵报警标志位
	
	VPEAlm					:BOOL;// 泵组报警
	
	VPEFasteStop			:BOOL;// 泵组快速停机标志位
	VPETailRowPre			:REAL:=0;// 尾排压力
	tcpConnected			:BOOL;// TCP 通讯链接成功
	
	busy					:BOOL;//泵组动作Busy状态
	done					:BOOL;//泵组动作Done状态
	opendone				:BOOL;//泵组动作伸出完成
	closedone				:BOOL;//泵组动作收回完成
	error					:BOOL;//泵组动作error状态
	errID					:UDINT;//泵组动作errID
	errTXT					:STRING(255):='';//泵组动作errTXT
	errWTXT					:WSTRING(255):="";//泵组动作errTXT 中文
END_VAR
	
VAR
	HMIItf					:VPEHMIStruts;//每个泵组对象都关联了一个HMI
	writeDataSize			:UINT;// 写入数据长度
	modebusAddr				:UINT;
	modebuseNum				:UINT;
	(*后续根据情况决定是否放到输入接口中；方便TCP远程通讯控制*)
	modeCtrl				:UINT:=2;// 控制模式（0：近控；2：远程；）
	CoModeCtrl				:UINT:=0;// 协调模式控制，默认0
	DryPumpCtrl				:UINT:=1;// 螺杆泵控制(0=关; 1=开; 2=待机)
	BoosterCtrl				:UINT:=1;// 罗茨泵控制(0=关; 1=开; 2=待机)
	FastStopCtrl			:UINT:=0;// 快速停机(0-自动停机; 1-快速停机)
	
	AccessModeStatus		:UINT:=0;// 控制状态（2：远程）
	DryPumpState			:DWORD:=100;// 螺杆泵状态（1=开; 0=关； 2=加减速）
	BoosteState				:DWORD:=100;// 罗茨泵状态（1=开; 0=关； 2=加减速）
	FastStopState			:DWORD:=0;// 快速停机已激活(0=否;1=是）
	
	DryPumpAlarm1			: DWORD:=0;// 螺杆泵报警1
	DryPumpAlarm2			: DWORD:=0;// 螺杆泵报警1
	
	BoosterAlarm1			: DWORD:=0;// 罗茨泵报警1
	BoosterAlarm2			: DWORD:=0;// 罗茨泵报警1
	
	runTON					: TON;
	
	openErrorDelayTon		:Ton;
	openDoneDelayTon		:Ton;
	closeErrorDelayTon		:Ton;
	closeDoneDelayTon		:Ton;
	
	extendTrigRAlc			:R_Trig;//上升沿触发
	runTimeClearR			:R_Trig;//上升沿触发
	openendTrigRAlc			:R_Trig;//上升沿触发
	
	singleControlR			:R_Trig;//上升沿触发
	singleControlF			:F_Trig;//上升沿触发
	
	openendTrigR1			:R_Trig;//上升沿触发
	closeractTrigR1			:R_Trig;//上升沿触发
	resetTrigR1				:R_Trig;//上升沿触发
	stopTrigR1				:R_Trig;//上升沿触发
	powerTrigR1				:R_Trig;//上升沿触发
	
	openStep				:UINT:=0;
	closeStep				:UINT:=0;
	errorStep				:UINT:=0;
	
	resetRelayTON			:TON;
	resetRelayTONTime		:TIME:=T#0.2S;
	
	notBusyMonitorDelayTon	:TON;//动作不切换时，延迟检测
	notBusyMonitorDelayTime :TIME:=T#2S;//动作不切换延迟检测时间
	firstPower			    :BOOL:=FALSE;//首次上电标志位
	
	AccRTrig:R_TRIG;//检测加速信号下降延
	AccTON:TON;//检测加速信号保持时间
	NormalRTrig:R_TRIG;//匀速上升沿
	DccRTrig:R_TRIG;// 检测减速信号下降延
	
	
	tcpStep						:UINT;				//处理步数
	tcpExcute					:BOOL;//
	tcpBusy						:BOOL;
	tcpDone						:BOOL;
	tcpError					:BOOL;
	tcpErrorID					:UINT;
	
	Timer1						:TON;
	
	tcpConnectedF_Trig			:F_TRIG;
	
	tcpipClient					:tcpipClientModule_EX;
	
	receveTemp:BOOL;
	
	tcpipSendDataBuff_Client	:ARRAY [1..12] OF BYTE;
	tcpipSendDataBuff_ClientTemp	:ARRAY [1..2] OF BYTE;
	tcpipRecDataBuff_Client	:ARRAY [1..100] OF BYTE;
	tcpipRecDataBuff_ClientTemp	:ARRAY [1..2] OF BYTE;
	tcpipRecDataBuff_clear	:ARRAY [1..100] OF BYTE;//数据清空
	bSendCondition:BOOL;
	tcpTimeOut:BOOL;//接收数据超时
	tcpRecError:BOOL;//接收数据错误
	tcpConnectR_Trig			:R_Trig;//初始连接上升沿
	tcpConnectF_Trig			:F_Trig;//初始连接下降沿
	VPEStateDate:POINTER TO VPETestStruts530;// 泵组运行、报警、停止等各种状态数据
	VPETempCurPowerDate:POINTER TO VPETestStruts540;// 泵组温度、速度、电流、功率等各种状态数据
	tcpComErrorTimes			:INT;
	tcpComErrorRestartT			:Ton;
	noteTON_P:tON;            // 操作提示标志位延时继电器
	noteTON_N:tON;            // 操作提示标志位延时继电器
	noteRTrig_P:R_TRIG;          // 操作提示
	noteRTrig_N:R_TRIG;          // 操作提示
	extRealayRtrig:R_TRIG;
	retRealayRtrig:R_TRIG;
END_VAR

Init_ACT();
Error_ACT();
Open_ACT();
Close_ACT();
Reset_ACT();
Error_ACT();
tcp_Act();

(*
触发缩回动作，成功触发返回TRUE，触发失败返回FALSE
*)
METHOD Act_Close : BOOL
VAR_INPUT
END_VAR
IF enable AND closeCondition THEN// AND NOT busy
	Act_Close:=close:=TRUE;
ELSE
	Act_Close:=FALSE;
END_IF
END_METHOD

(*
触发伸出动作，成功触发返回TRUE，触发失败返回FALSE
*)
METHOD Act_Open : BOOL
VAR_INPUT
END_VAR
IF enable AND openCondition THEN// AND NOT busy
	Act_Open:=open:=TRUE;
ELSE
	Act_Open:=FALSE;
END_IF
END_METHOD

(*
触发复位报警动作，成功触发返回TRUE，触发失败返回FALSE
*)
METHOD Act_Reset : BOOL
VAR_INPUT
END_VAR
Act_Reset:=reset:=TRUE;
END_METHOD

(*
触发停止输出动作，成功触发返回TRUE，触发失败返回FALSE
*)
METHOD Act_Stop : BOOL
VAR_INPUT
END_VAR
Act_Stop:=stop:=TRUE;
END_METHOD

(*
触发发送动作，成功触发返回TRUE，触发失败返回FALSE
*)
METHOD Act_TCPSend : BOOL
VAR_INPUT
END_VAR
IF TRUE THEN
	Act_TCPSend:=tcpExcute:=TRUE;
ELSE
	Act_TCPSend:=FALSE;
END_IF
END_METHOD

ACTION Close_ACT:
//分子泵--close 触发
IF close AND NOT closeCondition THEN
	note_open:=FALSE;
	note_close:=TRUE;
	NoteHMI.showFlag:=TRUE;
	NoteHMI.showText:='';
	NoteHMI.showText:=CONCAT(NoteHMI.showText,nameTXT);
	NoteHMI.showText:=CONCAT(NoteHMI.showText,' Close Condition Not Satisfied!');
END_IF
IF close AND enable AND closeCondition THEN// 
	note_open:=FALSE;
	note_close:=FALSE;
	busy:=TRUE;
	open:=FALSE;
	opendone:=FALSE;
	closedone:=FALSE;
	openStep:=0;
	closeStep:=10;
	Accing:=FALSE;
	Normal:=FALSE;
	Dccing:=FALSE;
	//errorStep:=0;
END_IF
close:=FALSE;

CASE closeStep OF
0:
	//ready
	
10:
	closeErrorDelayTon(IN:=FALSE);
	closeDoneDelayTon(IN:=FALSE);
	closeRelay:=TRUE;
	IF NOT openRelay AND AlmAprSw THEN
		closeStep:=40;
	ELSE
		closeStep:=20;
		openRelay:=FALSE;
	END_IF
20:
	closeErrorDelayTon(IN:=(NOT VPEFasteStop OR NOT openRelay),PT:=errorDelayTime);
	IF closeErrorDelayTon.Q THEN
		//done:=FALSE;
		opendone:=FALSE;
		closedone:=FALSE;
		errorStep:=2;
		Accing:=FALSE;
		Normal:=FALSE;
		Dccing:=FALSE;
		RETURN;
	END_IF
	IF (DryPumpState=2 OR BoosteState=2 OR VPEFasteStop) AND NOT openRelay THEN
		closeDoneDelayTon(IN:=(DryPumpState=2 OR BoosteState=2 OR VPEFasteStop) AND NOT openRelay,PT:=doneDelayTimeShortcloseract);
	END_IF
	IF closeDoneDelayTon.Q THEN
		Accing:=FALSE;
		Dccing:=TRUE;
		Normal:=FALSE;
		closeErrorDelayTon(IN:=FALSE);
		closeDoneDelayTon(IN:=FALSE);
		closeStep:=30;
	END_IF
30:
	closeErrorDelayTon(IN:=Dccing AND NOT openRelay,PT:=DCCMaxtime);
	IF closeErrorDelayTon.Q THEN
		//done:=FALSE;
		Accing:=FALSE;
		Dccing:=FALSE;
		Normal:=FALSE;
		opendone:=FALSE;
		closedone:=FALSE;
		closeStep:=60;
		openRelay:=FALSE;
		errorStep:=2;
		closeErrorDelayTon(IN:=FALSE);
	END_IF
	DccRTrig(CLK:=VPEFasteStop);
	IF DccRTrig.Q OR VPEFasteStop THEN
		closeStep:=40;
		Accing:=FALSE;
		Dccing:=FALSE;
		Normal:=FALSE;
		closeErrorDelayTon(IN:=FALSE);
	END_IF
40:
	IF NOT AccAprSw AND NOT VPEStart AND VPEFasteStop THEN
		busy:=FALSE;
		//done:=TRUE;
		opendone:=FALSE;
		closedone:=TRUE;
		errorStep:=0;
		closeStep:=50;
		IF NOT power (*AND NOT (CylinderType_Vacuum=cylinderType)*) THEN
			openRelay:=FALSE;
			closeRelay:=FALSE;
		END_IF
		closeRelay:=FALSE;
	ELSE
		busy:=FALSE;
		//done:=TRUE;
		opendone:=FALSE;
		closedone:=FALSE;
		errorStep:=3;
		closeStep:=60;
	END_IF
END_CASE
END_ACTION

ACTION Error_ACT:
CASE errorStep OF
	0:
		error:=FALSE;
		errID:=0;
		errTXT:='';
 (*
	1:
		error:=TRUE;
		errID:=errorID+errorStep;
		errTXT:=CONCAT(STR1:=nameTXT,STR2:=' Extend Error!');
		errWTXT:=WCONCAT(STR1:=TO_WSTRING(nameTXT),STR2:=" 伸出(打开)错误");
	2:
		error:=TRUE;
		errID:=errorID+errorStep;
		errTXT:=CONCAT(STR1:=nameTXT,STR2:=' Retract Error!');
		errWTXT:=WCONCAT(STR1:=TO_WSTRING(nameTXT),STR2:=" 缩回(关闭)错误");
		*)
	1..4:
		error:=TRUE;
		errID:=getErrID(errorStep);
		errTXT:=getErrTXT(errorStep);
		errWTXT:=getErrWTXT(errorStep);
END_CASE
END_ACTION

METHOD Get_Done_Close : BOOL
VAR_INPUT
END_VAR
Get_Done_Close:=closedone;
END_METHOD

METHOD Get_Done_Open : BOOL
VAR_INPUT
END_VAR
Get_Done_Open:=opendone;
END_METHOD

(*
触发发送动作，成功触发返回TRUE，触发失败返回FALSE
*)
METHOD Get_TCPSendBusy : BOOL
VAR_INPUT
END_VAR
Get_TCPSendBusy:=tcpDone;
END_METHOD

(*
触发发送动作，成功触发返回TRUE，触发失败返回FALSE
*)
METHOD Get_TCPSendDone : BOOL
VAR_INPUT
END_VAR
Get_TCPSendDone:=tcpDone;
END_METHOD

(*
触发发送动作，成功触发返回TRUE，触发失败返回FALSE
*)
METHOD Get_TCPSendError : BOOL
VAR_INPUT
END_VAR
Get_TCPSendError:=tcpError;
END_METHOD

METHOD getErrID : UDINT
VAR_INPUT
	errID					:UDINT;//取值范围1~2
END_VAR
VAR
	nErrID					:UDINT;
END_VAR
nErrID:=errorID+errID;

getErrID:=nErrID;
END_METHOD

METHOD getErrTXT : STRING(255)
VAR_INPUT
	errID					:UDINT;//取值范围1~2
END_VAR
VAR
	sErrTXT					:STRING(255);
END_VAR

CASE errID OF
	1:
		sErrTXT:=CONCAT(STR1:=nameTXT,STR2:=' Open Error!');
	2:
		sErrTXT:=CONCAT(STR1:=nameTXT,STR2:=' Close Error!');
	3:
		sErrTXT:=CONCAT(STR1:=nameTXT,STR2:=' NormalRun Error!');
	4:
		sErrTXT:=CONCAT(STR1:=nameTXT,STR2:=' CheckCondition Error!');
ELSE
	sErrTXT:=CONCAT(STR1:=nameTXT,STR2:='');
END_CASE
getErrTXT:=sErrTXT;
END_METHOD

METHOD getErrWTXT : WSTRING(255)
VAR_INPUT
	errID					:UDINT;//取值范围1~16
END_VAR
VAR
	sErrTXT					:WSTRING(255);
END_VAR

CASE errID OF
	1:
		sErrTXT:=WCONCAT(STR1:=TO_WSTRING(nameTXT),STR2:=" 分子泵启动错误");
	2:
		sErrTXT:=WCONCAT(STR1:=TO_WSTRING(nameTXT),STR2:=" 分子泵停止错误");
	3:
		sErrTXT:=WCONCAT(STR1:=TO_WSTRING(nameTXT),STR2:=" 分子泵正常运行出线异常情况");
	4:
		sErrTXT:=WCONCAT(STR1:=TO_WSTRING(nameTXT),STR2:=" 检测到条件异常，关机处理");
ELSE
	sErrTXT:=WCONCAT(STR1:=TO_WSTRING(nameTXT),STR2:="");
END_CASE
getErrWTXT:=sErrTXT;
END_METHOD

ACTION Init_ACT:
done:=(opendone OR closedone);
InitHMI_ACT();
manualCtrl_ACT();
stateMonitor();//状态监控


noteTON_P(IN:=note_open,PT:=T#0.1S);
noteRTrig_P(CLK:=noteTON_P.Q);
IF noteRTrig_P.Q THEN
//	gLog_Note.append_EX(noteWTXT_Open);
END_IF
noteTON_N(IN:=note_close,PT:=T#0.1S);
noteRTrig_N(CLK:=noteTON_N.Q);
IF noteRTrig_N.Q THEN
//	gLog_Note.append_EX(noteWTXT_close);
END_IF
extRealayRtrig(CLK:=openRelay);
IF extRealayRtrig.Q THEN
	HMIItf.singleControl:=TRUE;
END_IF
retRealayRtrig(CLK:=NOT openRelay);
IF retRealayRtrig.Q THEN
	HMIItf.singleControl:=FALSE;
END_IF
END_ACTION

ACTION InitHMI_ACT:
HMIItf.HMIEnable:=hmiEN;
HMIItf.enable:=enable;
HMIItf.done:=done;
HMIItf.busy:=busy;
HMIItf.error:=error OR VPEAlm;
HMIItf.errID:=UDINT_TO_DINT(errID);
HMIItf.errTXT:=errTXT;
HMIItf.openRelay:=openRelay;
HMIItf.power:=power;
HMIItf.nameTXT:=nameTXT;

HMIItf.AlmAprSw:=AlmAprSw;
HMIItf.AccAprSw:=AccAprSw;

HMIItf.runTime:=runTime;

//HMIItf.BoosterAlarm1:=BoosterAlarm1;
//HMIItf.BoosterAlarm2:=BoosterAlarm2;
HMIItf.BoosterCurrent:=DWORD_TO_REAL(BoosterCurrent)*0.1;
HMIItf.BoosterPower:=DWORD_TO_REAL(BoosterPower)*0.1;
HMIItf.BoosterSpeed:=DWORD_TO_REAL(BoosterSpeed)*0.1;
HMIItf.BoosterTemperature:=DWORD_TO_REAL(BoosterTemperature)*0.1;
HMIItf.BoosterStart:=bBooster;
HMIItf.BoosterError:=BoosterAlm;

//HMIItf.DryPumpAlarm1:=BoosterAlarm1;
//HMIItf.DryPumpAlarm2:=BoosterAlarm2;
HMIItf.DryPumpCurrent:=DWORD_TO_REAL(DryPumpCurrent)*0.1;
HMIItf.DryPumpPower:=DWORD_TO_REAL(DryPumpPower)*0.1;
HMIItf.DryPumpSpeed:=DWORD_TO_REAL(DryPumpSpeed)*0.1;
HMIItf.DryPumpTemperature:=DWORD_TO_REAL(DryPumpTemperature)*0.1;
HMIItf.DryPumpStart:=bDryPump;
HMIItf.DryPumpError:=DryPumpAlm;

HMIItf.Accing:=Accing;
HMIItf.Dccing:=Dccing;
HMIItf.Normal:=Normal;
HMIItf.tailrowPre:=VPETailRowPre;
HMIItf.opencondition:=openCondition;
HMIItf.closecondition:=closeCondition;
END_ACTION

ACTION ManualCtrl_ACT:
//HMI手动控制
IF hmiEN THEN
	extendTrigRAlc(CLK:=HMIItf.extendAndretract);
	IF extendTrigRAlc.Q THEN// AND NOT busy
		IF openRelay THEN// 如果启动继电器或全速，则认为已经已启动完毕
			close:=TRUE;
		END_IF
		IF NOT openRelay THEN
			open:=TRUE;
		END_IF
	END_IF
	
	singleControlR(CLK:=HMIItf.singleControltemp);
	openendTrigR1(CLK:=HMIItf.open);
	IF (openendTrigR1.Q OR (HMIItf.singleControltemp AND NOT HMIItf.singleControl)) THEN
		WarmHMI.showText:='';
		WarmHMI.showFlag:=TRUE;
		WarmHMI.showText:=CONCAT(WarmHMI.showText,'Are you sure you want to Open the ');
		WarmHMI.showText:=CONCAT(WarmHMI.showText,nameTXT);
		WarmHMI.showText:=CONCAT(WarmHMI.showText,' ?');
	END_IF
	IF WarmHMI.bOK AND NOT WarmHMI.showFlag AND FIND(WarmHMI.showText,nameTXT)>0 AND FIND(WarmHMI.showText,'Open')>0 THEN
		open:=TRUE;
		operatorLog.append(CONCAT(nameTXT,' Open'));
		close:=FALSE;
		HMIItf.singleControl:=NOT HMIItf.singleControl;
		WarmHMI.showText:='';
		WarmHMI.bOK:=FALSE;
		WarmHMI.showText:='';
	END_IF
	IF WarmHMI.bNO AND NOT WarmHMI.showFlag AND FIND(WarmHMI.showText,nameTXT)>0 AND FIND(WarmHMI.showText,'Open')>0 THEN
		WarmHMI.bNO:=FALSE;
		WarmHMI.showText:='';
	END_IF
	closeractTrigR1(CLK:=HMIItf.close);
	IF (closeractTrigR1.Q OR (HMIItf.singleControltemp AND HMIItf.singleControl)) THEN
		WarmHMI.showText:='';
		WarmHMI.showFlag:=TRUE;
		WarmHMI.showText:=CONCAT(WarmHMI.showText,'Are you sure you want to Close the ');
		WarmHMI.showText:=CONCAT(WarmHMI.showText,nameTXT);
		WarmHMI.showText:=CONCAT(WarmHMI.showText,' ?');
	END_IF
	IF WarmHMI.bOK AND NOT WarmHMI.showFlag AND FIND(WarmHMI.showText,nameTXT)>0 AND FIND(WarmHMI.showText,'Close')>0 THEN
		close:=TRUE;
		operatorLog.append(CONCAT(nameTXT,' Close'));
		open:=FALSE;
		HMIItf.singleControl:=NOT HMIItf.singleControl;
		WarmHMI.showText:='';
		WarmHMI.bOK:=FALSE;
		WarmHMI.showText:='';
	END_IF
	IF WarmHMI.bNO AND NOT WarmHMI.showFlag AND FIND(WarmHMI.showText,nameTXT)>0 AND FIND(WarmHMI.showText,'Close')>0 THEN
		WarmHMI.bNO:=FALSE;
		WarmHMI.showText:='';
	END_IF
	
	resetTrigR1(CLK:=HMIItf.reset);
	IF resetTrigR1.Q THEN// AND NOT busy
		reset:=TRUE;
	END_IF
	
	stopTrigR1(CLK:=HMIItf.stop);
	IF stopTrigR1.Q THEN// AND NOT busy
		stop:=TRUE;
	END_IF
	
	powerTrigR1(CLK:=HMIItf.power);
	IF powerTrigR1.Q THEN// AND NOT busy
		IF power THEN
			power:=FALSE;
		ELSE
			power:=TRUE;
		END_IF
	END_IF
END_IF
END_ACTION

ACTION Open_ACT:
//分子泵伸出--open 触发
IF open AND NOT openCondition THEN
	note_open:=TRUE;
	note_close:=FALSE;
	NoteHMI.showFlag:=TRUE;
	NoteHMI.showText:='';
	NoteHMI.showText:=CONCAT(NoteHMI.showText,nameTXT);
	NoteHMI.showText:=CONCAT(NoteHMI.showText,' Open Condition Not Satisfied!');
END_IF
IF open AND enable AND openCondition AND NOT BoosterAlm AND NOT DryPumpAlm AND NOT AlmAprSw AND openStep<20 AND NOT openRelay AND NOT VPEStart THEN// AND NOT busy
	note_open:=FALSE;
	note_close:=FALSE;
	busy:=TRUE;
	close:=FALSE;
	open:=FALSE;
	done:=FALSE;
	opendone:=FALSE;
	closedone:=FALSE;
	openStep:=10;
	closeStep:=0;
	
	Accing:=FALSE;
	Dccing:=FALSE;
	Normal:=FALSE;
END_IF
open:=FALSE;
runTimeClearR(CLK:=HMIItf.runTimeClear);
runTON(IN:=NOT error AND (openRelay OR VPEStart) AND AccAprSw AND NOT runTON.Q, PT:=T#36S);// 1小时计数一次,启动，无报错，且全速
IF runTON.Q AND runTime<999999999999999 AND NOT runTimeClearR.Q  THEN
	runTime:=runTime+1;
END_IF
IF runTimeClearR.Q THEN
	runTime:=0;
END_IF
//IF NOT openRelay AND NOT AccAprSw THEN// 计数清零
//	runTime:=0;
//END_IF
CASE openStep OF
0:
	//ready
	
10:
	openErrorDelayTon(IN:=FALSE);
	openDoneDelayTon(IN:=FALSE);
	AccTON(IN:=FALSE);
	openStep:=20;
	openRelay:=TRUE;
	closeRelay:=FALSE;
	tcpConnectedF_Trig(CLK:=FALSE);
20:
	(*
	通讯方式启动；不适用IO控制
	ModeCtrl:=2;
	CoModeCtrl:=0;
	DryPumpCtrl:=1;
	BoosterCtrl:=1;*)
	openErrorDelayTon(IN:=VPEFasteStop,PT:=T#30S);// 检测停止信号
	IF openErrorDelayTon.Q THEN
		opendone:=FALSE;
		closedone:=FALSE;
		openStep:=60;
		openRelay:=FALSE;
		errorStep:=1;
		openErrorDelayTon(IN:=FALSE);
		Accing:=FALSE;
		Normal:=FALSE;
		Dccing:=FALSE;
	ELSE
		IF NOT VPEFasteStop THEN
			openErrorDelayTon(IN:=FALSE);
			openStep:=30;
		END_IF
	END_IF
	
30:
	AccTON(IN:=((DryPumpState=2 OR BoosteState=2) OR (DryPumpState=1 AND BoosteState=1)) AND openRelay AND NOT VPEFasteStop,PT:=T#5S);// 检测虚假加速信号
	AccRTrig(CLK:=(DryPumpState=2 OR BoosteState=2));
	IF AccRTrig.Q OR AccTON.Q THEN
		Accing:=TRUE;
		Normal:=FALSE;
		Dccing:=FALSE;
		openStep:=40;
		openErrorDelayTon(IN:=FALSE);
	END_IF
	//状态实时检测
	IF (AlmAprSw OR VPEAlm) AND openRelay THEN//只要报错；启动线圈启动，强锁启动信号
		openRelay:=FALSE;
		close:=TRUE;
		stop:=TRUE;
		openStep:=60;/////
		errorStep:=3;
		Accing:=FALSE;
		Dccing:=FALSE;
		Normal:=FALSE;
	END_IF
40:
	openErrorDelayTon(IN:=NOT VPEStart ,PT:=ACCMaxtime);//检测预热信号
	IF openErrorDelayTon.Q THEN
		//done:=FALSE;
		opendone:=FALSE;
		closedone:=FALSE;
		openStep:=60;
		openRelay:=FALSE;
		errorStep:=1;
		openErrorDelayTon(IN:=FALSE);
		Accing:=FALSE;
		Normal:=FALSE;
		Dccing:=FALSE;
	END_IF
	IF VPEStart THEN
		Accing:=FALSE;
		Dccing:=FALSE;
		Normal:=TRUE;
		busy:=FALSE;
		//done:=TRUE;
		opendone:=TRUE;
		closedone:=FALSE;
		openStep:=50;
		IF NOT power (*AND NOT (CylinderType_Vacuum=cylinderType)*) THEN
			openRelay:=FALSE;
			closeRelay:=FALSE;
		END_IF
	END_IF
50:
	IF real_TimeMonitor THEN
		//启动实时检测
		IF NOT openRelay THEN//启动后，检测到关信号
			errorStep:=1;
			openRelay:=FALSE;
			openStep:=60;
		END_IF
		IF (AlmAprSw OR VPEAlm) AND openRelay THEN//只要报错；启动线圈启动，强锁启动信号
			openRelay:=FALSE;
			close:=TRUE;
			stop:=TRUE;
			openStep:=60;/////
			errorStep:=3;
		END_IF
		tcpConnectedF_Trig(CLK:=tcpConnected);//通讯掉线
		IF tcpConnectedF_Trig.Q THEN
			tcpConnectedF_Trig(CLK:=FALSE);
			errorStep:=4;//通讯异常
		END_IF
	END_IF
60:
	;//报错
END_CASE
END_ACTION

ACTION Reset_ACT:
IF reset THEN
	IF NOT power THEN
		openRelay:=FALSE;
		closeRelay:=FALSE;
	END_IF
	IF error THEN
		busy:=FALSE;
	END_IF
	//done:=FALSE;
	errorStep:=0;
	resetRelay:=TRUE;
	
	reset:=FALSE;
	note_open:=FALSE;
	note_close:=FALSE;
END_IF
resetRelayTON(IN:=resetRelay , PT:=resetRelayTONTime);
IF resetRelayTON.Q THEN
	resetRelay:=FALSE;
END_IF

IF stop THEN
	stop:=FALSE;
	openRelay:=FALSE;
	closeRelay:=FALSE;
	//无自锁检测说法，直接停
	openStep:=0;
	closeStep:=0;
	busy:=FALSE;
END_IF
END_ACTION

ACTION stateMonitor:
IF tcpConnected THEN//状态监控
	bDryPump:=DryPumpState=1;//等于1 启动
	bBooster:=BoosteState=1;//等于1 启动
	VPEStart:=bDryPump AND bBooster AND AccAprSw;
	DryPumpAlm:=(DryPumpAlarm1<>0 AND DryPumpAlarm2<>0) OR tcpError ;
	BoosterAlm:=(BoosterAlarm1<>0 AND BoosterAlarm2<>0) OR tcpError;
	VPEAlm:=DryPumpAlm OR BoosterAlm OR AlmAprSw (*OR tcpError*);
	VPEFasteStop:=FastStopState=0 OR (DryPumpState=0 AND BoosteState=0);//快速停机标志位
ELSE
	VPEAlm:=AlmAprSw OR tcpError;
END_IF
IF enabletcp AND errorStep=4 AND tcpConnected THEN
	errorStep:=0;
END_IF
IF VPEAlm AND openRelay THEN
	close:=TRUE;
	stop:=TRUE;
	openRelay:=FALSE;
END_IF
END_ACTION

ACTION tcp_Act:
tcpipClient(
		sSrvNetId:= , 
		sRemoteHost:=sHost , 
		nRemotePort:=nPort , 
		bStartConnect:=bEnable , 
		tcpipSDataLen:=SIZEOF(tcpipSendDataBuff_Client) , 
		tcpipSData:=ADR(tcpipSendDataBuff_Client) , 
		bSend:= , 
		tcpipRecDataLen:=SIZEOF(tcpipRecDataBuff_Client) , 
		tcpipRecData:=ADR(tcpipRecDataBuff_Client) , 
		bConnected=>tcpConnected , 
		bSendBusy=> , 
		bRecData=> );
	bSendCondition:=tcpipClient.bConnected AND NOT tcpipClient.bSendBusy;
	tcpConnectR_Trig(CLK:=tcpConnected);
	tcpConnectF_Trig(CLK:=tcpConnected);
	IF tcpConnectR_Trig.Q THEN
		gLog.append(CONCAT(nameTXT, ' has been connected'));
		tcpStep:=0;
		tcpBusy:=FALSE;
		tcpDone:=FALSE;
		tcpError:=FALSE;
		tcpTimeOut:=FALSE;
		tcpRecError:=FALSE;
		tcpExcute:=TRUE;
		tcpComErrorTimes:=0;
	END_IF
	IF tcpConnectF_Trig.Q THEN
		gLog.append(CONCAT(nameTXT, ' has been disconnected'));
		IF enabletcp THEN
			tcpStep:=0;
			tcpBusy:=FALSE;
			tcpDone:=FALSE;
			tcpError:=TRUE;
			tcpTimeOut:=FALSE;
			tcpRecError:=FALSE;
		ELSE
			tcpStep:=0;
			tcpBusy:=FALSE;
			tcpDone:=FALSE;
			tcpError:=FALSE;
			tcpTimeOut:=FALSE;
			tcpRecError:=FALSE;
		END_IF
	END_IF
	IF  tcpipClient.bRecData THEN//接收完成
		receveTemp:=TRUE;
	END_IF
CASE tcpStep OF
	0:
	IF enabletcp AND tcpExcute THEN
		tcpExcute:=FALSE;
		IF NOT tcpBusy AND tcpConnected THEN
			tcpStep:=10;
			tcpBusy:=TRUE;
			tcpDone:=FALSE;
			tcpError:=FALSE;
			tcpTimeOut:=FALSE;
			tcpRecError:=FALSE;
			//复位
		END_IF
	END_IF
	Timer1(IN:= FALSE);
	;
	10:
		receveTemp:=FALSE;
		tcpipSendDataBuff_Client[1]:=0;
		tcpipSendDataBuff_Client[2]:=0;
		tcpipSendDataBuff_Client[3]:=0;
		tcpipSendDataBuff_Client[4]:=0;
		tcpipSendDataBuff_Client[5]:=0;
		tcpipSendDataBuff_Client[6]:=16#06;
		tcpipSendDataBuff_Client[7]:=UINT_TO_BYTE(slaveID);
		tcpipSendDataBuff_Client[8]:=16#03;
		modebusAddr:=530;
		MEMMOVE(ADR(tcpipSendDataBuff_ClientTemp[1]),ADR(modebusAddr),2);
		tcpipSendDataBuff_Client[9]:=tcpipSendDataBuff_ClientTemp[2];
		tcpipSendDataBuff_Client[10]:=tcpipSendDataBuff_ClientTemp[1];
		modebuseNum:=10;
		MEMMOVE(ADR(tcpipSendDataBuff_ClientTemp[1]),ADR(modebuseNum),2);
		tcpipSendDataBuff_Client[11]:=tcpipSendDataBuff_ClientTemp[2];
		tcpipSendDataBuff_Client[12]:=tcpipSendDataBuff_ClientTemp[1];
		
		tcpStep:=100;
		Timer1(IN:= FALSE);
	100:
		tcpipClient.bSend:=TRUE;
		tcpStep:=tcpStep+20;
	110:
		tcpStep:=tcpStep+10;
	120:
		Timer1(IN:= NOT timer1.q, PT:=T#3000MS);
		IF Timer1.Q THEN
			tcpipClient.bSend:=FALSE;
			tcpStep:=6000;
			tcpTimeOut:=TRUE;
			Timer1(IN:= FALSE);
			RETURN;
		END_IF
		//接收数据
		IF  receveTemp THEN//接收完成
			tcpipClient.bSend:=FALSE;
			Timer1(IN:= FALSE);
			receveTemp:=FALSE;
			tcpStep:=200;
		END_IF
	200://数据处理
		tcpStep:=tcpStep+10;
	210:
		IF  tcpipRecDataBuff_Client[1]=tcpipSendDataBuff_Client[1] AND  tcpipRecDataBuff_Client[2]=tcpipSendDataBuff_Client[2] AND  
			tcpipRecDataBuff_Client[3]=tcpipSendDataBuff_Client[3] AND  tcpipRecDataBuff_Client[4]=tcpipSendDataBuff_Client[4] AND  
			tcpipRecDataBuff_Client[7]=tcpipSendDataBuff_Client[7] THEN//数据判断,反馈数据与发送数据匹配无误
				
			DryPumpState:=BYTE_TO_WORD(tcpipRecDataBuff_Client[10])*256+BYTE_TO_WORD(tcpipRecDataBuff_Client[11]);
			BoosteState:=BYTE_TO_WORD(tcpipRecDataBuff_Client[12])*256+BYTE_TO_WORD(tcpipRecDataBuff_Client[13]);
			FastStopState:=BYTE_TO_WORD(tcpipRecDataBuff_Client[14])*256+BYTE_TO_WORD(tcpipRecDataBuff_Client[15]);
			DryPumpAlarm1:=BYTE_TO_WORD(tcpipRecDataBuff_Client[18])*256+BYTE_TO_WORD(tcpipRecDataBuff_Client[19]);
			BoosterAlarm1:=BYTE_TO_WORD(tcpipRecDataBuff_Client[20])*256+BYTE_TO_WORD(tcpipRecDataBuff_Client[21]);
			DryPumpAlarm2:=BYTE_TO_WORD(tcpipRecDataBuff_Client[22])*256+BYTE_TO_WORD(tcpipRecDataBuff_Client[23]);
			BoosterAlarm2:=BYTE_TO_WORD(tcpipRecDataBuff_Client[24])*256+BYTE_TO_WORD(tcpipRecDataBuff_Client[25]);
			DryPumpSpeed:=BYTE_TO_WORD(tcpipRecDataBuff_Client[26])*256+BYTE_TO_WORD(tcpipRecDataBuff_Client[27]);
			BoosterSpeed:=BYTE_TO_WORD(tcpipRecDataBuff_Client[28])*256+BYTE_TO_WORD(tcpipRecDataBuff_Client[29]);
			tcpipRecDataBuff_Client:=tcpipRecDataBuff_clear;
			tcpStep:=tcpStep+10;
		ELSE//数据接线错误
			tcpStep:=6000;
			tcpRecError:=TRUE;
		END_IF
	220:
		//数据转换
		tcpTimeOut:=FALSE;
		tcpRecError:=FALSE;
		tcpStep:=300;
		Timer1(IN:= FALSE);
	;
	300:
		tcpError:=FALSE;
		tcpStep:=400;
	400:
		Timer1(IN:= NOT timer1.q, PT:=T#2000MS);
		IF Timer1.Q THEN
			Timer1(IN:= FALSE);
			tcpStep:=tcpStep+10;
		END_IF
	410://第二次轮询
		receveTemp:=FALSE;
		tcpipSendDataBuff_Client[1]:=0;
		tcpipSendDataBuff_Client[2]:=0;
		tcpipSendDataBuff_Client[3]:=0;
		tcpipSendDataBuff_Client[4]:=0;
		tcpipSendDataBuff_Client[5]:=0;
		tcpipSendDataBuff_Client[6]:=16#06;
		tcpipSendDataBuff_Client[7]:=UINT_TO_BYTE(slaveID);
		tcpipSendDataBuff_Client[8]:=16#03;
		modebusAddr:=540;
		MEMMOVE(ADR(tcpipSendDataBuff_ClientTemp[1]),ADR(modebusAddr),2);
		tcpipSendDataBuff_Client[9]:=tcpipSendDataBuff_ClientTemp[2];
		tcpipSendDataBuff_Client[10]:=tcpipSendDataBuff_ClientTemp[1];
		modebuseNum:=10;
		MEMMOVE(ADR(tcpipSendDataBuff_ClientTemp[1]),ADR(modebuseNum),2);
		tcpipSendDataBuff_Client[11]:=tcpipSendDataBuff_ClientTemp[2];
		tcpipSendDataBuff_Client[12]:=tcpipSendDataBuff_ClientTemp[1];
		
		tcpStep:=500;
		Timer1(IN:= FALSE);
	500:
		tcpipClient.bSend:=TRUE;
		tcpStep:=tcpStep+20;
	510:
		tcpStep:=tcpStep+10;
	520:
		Timer1(IN:= NOT timer1.q, PT:=T#3000MS);
		IF Timer1.Q THEN
			tcpipClient.bSend:=FALSE;
			tcpStep:=6000;
			tcpTimeOut:=TRUE;
			Timer1(IN:= FALSE);
			RETURN;
		END_IF
		//接收数据
		IF  receveTemp THEN//接收完成
			tcpipClient.bSend:=FALSE;
			Timer1(IN:= FALSE);
			receveTemp:=FALSE;
			tcpStep:=600;
		END_IF
	600://数据处理
		tcpStep:=tcpStep+10;
	610:
		IF  tcpipRecDataBuff_Client[1]=tcpipSendDataBuff_Client[1] AND  tcpipRecDataBuff_Client[2]=tcpipSendDataBuff_Client[2] AND  
			tcpipRecDataBuff_Client[3]=tcpipSendDataBuff_Client[3] AND  tcpipRecDataBuff_Client[4]=tcpipSendDataBuff_Client[4] AND  
			tcpipRecDataBuff_Client[7]=tcpipSendDataBuff_Client[7] THEN//数据判断,反馈数据与发送数据匹配无误
			DryPumpTemperature:=BYTE_TO_WORD(tcpipRecDataBuff_Client[10])*256+BYTE_TO_WORD(tcpipRecDataBuff_Client[11]);
			BoosterTemperature:=BYTE_TO_WORD(tcpipRecDataBuff_Client[14])*256+BYTE_TO_WORD(tcpipRecDataBuff_Client[15]);
			DryPumpPower:=BYTE_TO_WORD(tcpipRecDataBuff_Client[18])*256+BYTE_TO_WORD(tcpipRecDataBuff_Client[19]);
			BoosterPower:=BYTE_TO_WORD(tcpipRecDataBuff_Client[20])*256+BYTE_TO_WORD(tcpipRecDataBuff_Client[21]);
			DryPumpCurrent:=BYTE_TO_WORD(tcpipRecDataBuff_Client[22])*256+BYTE_TO_WORD(tcpipRecDataBuff_Client[23]);
			BoosterCurrent:=BYTE_TO_WORD(tcpipRecDataBuff_Client[24])*256+BYTE_TO_WORD(tcpipRecDataBuff_Client[25]);
			tcpStep:=tcpStep+10;
			tcpipRecDataBuff_Client:=tcpipRecDataBuff_clear;
		ELSE//数据接线错误
			tcpStep:=6000;
			tcpRecError:=TRUE;
		END_IF
	620:
		tcpTimeOut:=FALSE;
		tcpRecError:=FALSE;
		tcpComErrorTimes:=0;
		tcpStep:=700;
	700:
		Timer1(IN:= NOT timer1.q, PT:=T#2000MS);
		IF Timer1.Q THEN
			Timer1(IN:= FALSE);
			tcpStep:=tcpStep+10;
		END_IF
	710:
		tcpStep:=800;
	;
	800:
		receveTemp:=FALSE;
		tcpipSendDataBuff_Client[1]:=0;
		tcpipSendDataBuff_Client[2]:=0;
		tcpipSendDataBuff_Client[3]:=0;
		tcpipSendDataBuff_Client[4]:=0;
		tcpipSendDataBuff_Client[5]:=0;
		tcpipSendDataBuff_Client[6]:=16#06;
		tcpipSendDataBuff_Client[7]:=UINT_TO_BYTE(slaveID);
		tcpipSendDataBuff_Client[8]:=16#03;
		modebusAddr:=552;
		MEMMOVE(ADR(tcpipSendDataBuff_ClientTemp[1]),ADR(modebusAddr),2);
		tcpipSendDataBuff_Client[9]:=tcpipSendDataBuff_ClientTemp[2];
		tcpipSendDataBuff_Client[10]:=tcpipSendDataBuff_ClientTemp[1];
		modebuseNum:=1;
		MEMMOVE(ADR(tcpipSendDataBuff_ClientTemp[1]),ADR(modebuseNum),2);
		tcpipSendDataBuff_Client[11]:=tcpipSendDataBuff_ClientTemp[2];
		tcpipSendDataBuff_Client[12]:=tcpipSendDataBuff_ClientTemp[1];
		
		tcpStep:=tcpStep+10;
		Timer1(IN:= FALSE);
	810:
		tcpipClient.bSend:=TRUE;
		tcpStep:=tcpStep+20;
	820:
		tcpStep:=tcpStep+10;
	830:
		Timer1(IN:= NOT timer1.q, PT:=T#3000MS);
		IF Timer1.Q THEN
			tcpipClient.bSend:=FALSE;
			tcpStep:=6000;
			tcpTimeOut:=TRUE;
			Timer1(IN:= FALSE);
			RETURN;
		END_IF
		//接收数据
		IF  receveTemp THEN//接收完成
			tcpipClient.bSend:=FALSE;
			Timer1(IN:= FALSE);
			receveTemp:=FALSE;
			tcpStep:=900;
		END_IF
	900://数据处理
		tcpStep:=tcpStep+10;
	910:
		IF  tcpipRecDataBuff_Client[1]=tcpipSendDataBuff_Client[1] AND  tcpipRecDataBuff_Client[2]=tcpipSendDataBuff_Client[2] AND  
			tcpipRecDataBuff_Client[3]=tcpipSendDataBuff_Client[3] AND  tcpipRecDataBuff_Client[4]=tcpipSendDataBuff_Client[4] AND  
			tcpipRecDataBuff_Client[7]=tcpipSendDataBuff_Client[7] THEN//数据判断,反馈数据与发送数据匹配无误
				
			VPETailRowPre:=BYTE_TO_WORD(tcpipRecDataBuff_Client[10])*256+BYTE_TO_WORD(tcpipRecDataBuff_Client[11]);

			tcpipRecDataBuff_Client:=tcpipRecDataBuff_clear;
			tcpStep:=tcpStep+10;
		ELSE//数据接线错误
			tcpStep:=6000;
			tcpRecError:=TRUE;
		END_IF
	920:
		//数据转换
		tcpTimeOut:=FALSE;
		tcpRecError:=FALSE;
		tcpStep:=tcpStep+10;
		Timer1(IN:= FALSE);
	;
	930:
		Timer1(IN:= NOT timer1.q, PT:=T#2000MS);
		IF Timer1.Q THEN
			Timer1(IN:= FALSE);
			tcpStep:=tcpStep+10;
			tcpError:=FALSE;
		END_IF
	940:
		tcpStep:=10;
	5000://done
		tcpBusy:=FALSE;
		tcpDone:=TRUE;
		tcpError:=FALSE;
		tcpStep:=0;
		tcpipRecDataBuff_Client:=tcpipRecDataBuff_clear;
	;
	6000://error
		tcpDone:=FALSE;
		tcpError:=TRUE;
		tcpComErrorTimes:=tcpComErrorTimes+1;
		tcpComErrorRestartT(IN:=tcpComErrorTimes>30 AND NOT tcpComErrorRestartT.Q ,PT:=T#2S);
		IF tcpComErrorRestartT.Q THEN
			tcpComErrorTimes:=0;
			tcpStep:=0;
			tcpBusy:=FALSE;
			bEnable:=TRUE;
			RETURN;
		END_IF
		IF tcpComErrorTimes>10 THEN
			bEnable:=FALSE;
			RETURN;
		END_IF
		tcpipRecDataBuff_Client:=tcpipRecDataBuff_clear;
		tcpStep:=10;
	;
	
END_CASE
END_ACTION

ACTION VersionLog:
(*
版本: V1.0.0.0
说明:
	1. 首个版本
	2. 含普通分子泵\泵组类型的控制
	3. 可配置是否有到位信号, 以及到位稳定时间
(--------------------------------------------------)
新版本: V1.0.1.0
更新时间: 2019/11/20 19:00
更新说明:
	1. 优化编写方式
	2. 修改错误编码起始位，现改为从1开始
(--------------------------------------------------)
新版本: V1.0.1.1
更新时间: 2020/03/23 23:00
更新说明:
	1. 优化报错方式
	2. 增加伸出、缩回、复位和停止触发函数
(--------------------------------------------------)
新版本: V1.0.1.2
更新时间: 2020/04/22 09:50
更新说明:
	1. 增加中文报警输出
(--------------------------------------------------)
新版本: V1.0.1.3
更新时间: 2020/09/16
更新说明:
	1. 开放错误ID、错误文本信息获取接口
(--------------------------------------------------)
新版本: V1.0.1.4
更新时间: 2020/10/06
更新说明:
	1. 移除控制模式变量，增加HMI启用条件
	2. 增加外部获取伸出缩回完成信号接口函数
(--------------------------------------------------)
新版本: V1.0.1.5
更新时间: 2020/10/14
更新说明:
	1. 优化代码
(--------------------------------------------------)
新版本: V2.0.1.0
更新时间: 2023/11/17
更新说明:
	1. 分子泵控制独立
(--------------------------------------------------)


*)
END_ACTION

END_FUNCTION_BLOCK

// ---- POUs/BaseModule/TcpIpModule_EX/clientModule_EX/tcpipClientModule_EX.TcPOU
//可实现TCPIP Client 数据的收发
FUNCTION_BLOCK tcpipClientModule_EX
VAR_INPUT
//Connect
	sSrvNetId			:T_AmsNetId:='';
	sRemoteHost			:STRING(20):='127.0.0.1';//服务器的IP地址
	nRemotePort			:UDINT:=6000;//服务器的端口号
	bStartConnect		:BOOL:=TRUE;//可实现外部控制客户端的打开和关闭
//Send
	tcpipSDataLen		:UDINT;//待发送数据长度--外部传递进来
	tcpipSData			:POINTER TO BYTE;//待发送数据源----外部以指针的形式传递进来
	bSend				:BOOL:=FALSE;//数据发送触发信号
//Receive
	tcpipRecDataLen		:UDINT;//已接收数据长度--外部传递进来
	tcpipRecData		:POINTER TO BYTE;//已接收数据源--外部以指针的形式传递进来(ADR函数)
END_VAR

VAR_OUTPUT
//Connect
	bConnected			:BOOL:=FALSE;//表示连接状态
//Send
	bSendBusy			:BOOL:=FALSE;//数据发送中
//Receive
	bRecData			:BOOL:=FALSE;//数据接收有效信号, 上升沿有效
END_VAR

VAR
//Connect
	conStep				:UINT:=0;
	connectFB			:FB_SocketConnect;
	hSocket				:T_HSOCKET;
	conDelayTime		:TIME:=T#500MS;
	conDelayTon			:TON;
	conCheckTime		:TIME:=T#500MS;
	conCheckTon			:TON;
//Close
	closeFB				:FB_SocketClose;
//Receive
	recStep				:UINT:=0;
	receiveFB			:FB_SocketReceive;
	recDelayTime		:TIME:=T#1S;
	recDelayTon			:TON;
//Send
	sendStep			:UINT:=0;
	sendFB				:FB_SocketSend;
	sendDataTempLen		:UDINT;//待发送数据缓存 长度
	sendDataTemp		:POINTER TO BYTE;//待发送数据缓存
END_VAR

connect();
receive();
send();
closeFB(
	sSrvNetId:=sSrvNetId,
	hSocket:=,
	bExecute:=FALSE);

METHOD ascii2String : STRING(g_nMaxByte_Client)
VAR_INPUT
	byteArr:ARRAY [1..g_nMaxByte_Client] OF BYTE;
END_VAR
VAR
	i:UINT;
	strTemp:STRING(g_nMaxByte_Client);
END_VAR
FOR i:=1 TO g_nMaxByte_Client DO
	strTemp:=concat(strTemp,F_ToCHR(c:=byteArr[i]));
END_FOR
ascii2String:=strTemp;
END_METHOD

METHOD PRIVATE close : BOOL
VAR_INPUT
END_VAR
//关闭hSocket这个端口的连接
closeFB(
	sSrvNetId:=sSrvNetId,
	hSocket:=hSocket, 
	bExecute:=TRUE, 			//TCP/IP端口关闭的执行位
	tTimeout:=,
	bBusy=>,
	bError=>,
	nErrId=>);
closeFB(
	sSrvNetId:=sSrvNetId,
	hSocket:=,
	bExecute:=FALSE);
hSocket.handle:=0;
bConnected:=FALSE;
END_METHOD

METHOD PRIVATE connect : BOOL
VAR_INPUT
END_VAR

VAR
END_VAR

CASE conStep OF
0:
	IF bStartConnect THEN
		IF bConnected THEN
			RETURN;
		END_IF
		close();
		connectFB(sSrvNetId:=sSrvNetId,bExecute:= FALSE,hSocket=> hSocket);
		conStep:=conStep+1;
	ELSE
		conStep:=3;
	END_IF

1:
	connectFB(
		sSrvNetId:=sSrvNetId,
		sRemoteHost:=sRemoteHost,
		nRemotePort:=nRemotePort,
		bExecute:=TRUE,
		hSocket=>hSocket,
		nErrId=>);
	IF NOT connectFB.bBusy THEN
		IF connectFB.bError OR hSocket.handle=0 THEN
			close();
			conStep:=conStep+1;
		ELSE
			connectFB(sSrvNetId:=sSrvNetId,bExecute:= FALSE);
			conStep:=50;						
		END_IF
	END_IF
	conDelayTon(IN:=FALSE);

2://delay
	conDelayTon(IN:=NOT conDelayTon.Q ,PT:=conDelayTime);
	IF conDelayTon.Q THEN
		conDelayTon(in:=FALSE);
		conStep:=conStep+1;
	END_IF

3://close socket
	close();
	conStep:=conStep+1;

4:
	IF hSocket.handle<>0 THEN
		//conStep:=conStep-1;
		conStep:=conStep+1;
	ELSE
		conStep:=conStep+1;
	END_IF
	
5://try again
	conStep:=0;

50:
	conDelayTon(IN:=NOT conDelayTon.Q ,PT:=T#1500MS);
	IF conDelayTon.Q THEN
		conDelayTon(in:=FALSE);
		bConnected:=TRUE;
		conStep:=100;
	END_IF
	conCheckTon(in:=FALSE);
	
100://check connect status//done do nothing
	conCheckTon(IN:=NOT bConnected OR NOT bStartConnect,PT:=conCheckTime);//NOT conCheckTon.Q
	IF conCheckTon.Q THEN			
		conStep:=0;
		conCheckTon(in:=FALSE);
	END_IF

END_CASE
END_METHOD

METHOD PRIVATE receive : BOOL
VAR_INPUT
END_VAR
VAR
	recDataClear		:POINTER TO BYTE;//已接收数据源--外部以指针的形式传递进来(ADR函数)
END_VAR
	
CASE recStep OF
0:
	IF hSocket.handle>0 THEN
		recStep:=10;
	END_IF
10:
	bRecData:=FALSE;
	receiveFB(
		sSrvNetId:=sSrvNetId,
		hSocket:=hSocket,
		cbLen:= tcpipRecDataLen,
		pDest:= tcpipRecData,
		bExecute:= TRUE,
		tTimeout:=T#1S,
		bBusy=>,
		bError=>,
		nErrId=>,
		nRecBytes=>);
	
	IF (NOT receiveFB.bBusy) THEN
		recStep:=20;
	END_IF
20:
	receiveFB(sSrvNetId:=sSrvNetId,hSocket:=hSocket,bExecute :=FALSE);
	IF (NOT receiveFB.bBusy) THEN
		IF (receiveFB.bError) THEN
			close();
			recStep:=110;
		ELSE
			IF ReceiveFB.nRecBytes>0 THEN
				tcpipRecData:=recDataClear;//清空缓存数据
				
				bRecData:=TRUE;
			END_IF
			recStep:=10;//Re-Receive
		END_IF
	END_IF

110:
	recDelayTon(IN:=FALSE);
	recStep:=recStep+10;
120:
	recDelayTon(IN:=NOT recDelayTon.Q ,PT:=recDelayTime);
	IF recDelayTon.Q THEN
		recDelayTon(IN:=FALSE);
		recStep:=recStep+10;
	END_IF
130:
	recStep:=0;
END_CASE
END_METHOD

METHOD PRIVATE send : BOOL
VAR_INPUT
END_VAR
VAR
END_VAR

CASE sendStep OF
0:
	IF bConnected THEN
		bSendBusy:=FALSE;
		sendFB(sSrvNetId:=sSrvNetId,hSocket:=hSocket,bExecute:=FALSE);
		IF bSend THEN
			sendStep:=10;
			sendDataTempLen:=tcpipSDataLen;
			sendDataTemp:=tcpipSData;
			bSendBusy:=TRUE;
			bSend:=FALSE;
		END_IF
	END_IF
10:
	sendFB(
		sSrvNetId:=sSrvNetId,
		hSocket:=hSocket,
		cbLen:= sendDataTempLen,
		pSrc:= sendDataTemp,
		bExecute:= TRUE,
		tTimeout:=T#1S,
		bBusy=>,
		bError=>,
		nErrId=>);
	
	IF NOT sendFB.bBusy THEN
		sendStep:=sendStep+10;
	END_IF
20:
	sendStep:=sendStep+10;
30:
	bSendBusy:=FALSE;
	bSend:=FALSE;
	sendStep:=0;
END_CASE
END_METHOD

METHOD string2ASCII : ARRAY [1..g_nMaxByte_Client] OF BYTE
VAR_INPUT
	str:STRING(g_nMaxByte_Client);
END_VAR
VAR
	i:DINT;
	byteTemp:ARRAY [1..g_nMaxByte_Client] OF BYTE;
	strB:STRING(1);
	strTemp:STRING(g_nMaxByte_Client);
END_VAR
strTemp:=str;
FOR i:=1 TO g_nMaxByte_Client DO
	strB:=LEFT(strTemp,1);
	strTemp:=DELETE(strTemp,1,1);
	byteTemp[i]:=F_ToASC(str:=strB);
END_FOR
string2ASCII:=byteTemp;
END_METHOD

ACTION VersionLog:
(*
版本: V1.0.0.0
说明:
	1. 首个版本
(**************************************************)
版本: V1.0.0.1
说明:
	1. 更新close函数，关闭连接后清零连接句柄
(**************************************************)
*)
END_ACTION

END_FUNCTION_BLOCK

// ---- POUs/BaseModule/ActionModule/PendulumValveModule/PVModule.TcPOU
(*
--报错编号0: 无报错
--报错编号1: open Error
--报错编号2: close Error
*)
FUNCTION_BLOCK PVModule
VAR_IN_OUT
	WarmHMI					:WARMStruct;
	NoteHMI					:NoteStruct;
	operatorLog				:printLogModule_EX;
	opencondition_INOUT		:BOOL;
END_VAR
VAR_INPUT
	HMIItf						:PVModuleHMI;//每个PV对象都关联了一个HMI
	pvType						:PVType:=PVType_Default;// 设置PV的类型, 可通过该变量修改为其他品牌的PV阀门
	controlMode					:PVControlMOD:=PVControl_Default;
	real_TimeMonitor			:BOOL:=TRUE;//实时状态检测
	
	openRemOK					:BOOL:=FALSE;// 腔体无传感器真空记忆标记
	open						:BOOL:=FALSE;//打开触发信号
	openCondition				:BOOL:=TRUE;//打开启停条件
	close						:BOOL:=FALSE;// 关闭触发信号
	closeCondition				:BOOL:=TRUE;// 关闭启停条件
	mode						:BOOL:=FALSE;// 模式切换触发信号
	modeCondition				:BOOL:=TRUE;// 打开模式切换条件
	config						:BOOL:=FALSE;// 配置模式触发信号
	configCondition				:BOOL:=TRUE;// 配置模式触发条件
	reset						:BOOL:=FALSE;//复位信号
	readCondition				:BOOL:=TRUE; // 循环读取
	stop						:BOOL:=FALSE;//停止信号
	power						:BOOL:=TRUE;//PV动作后是否关闭继电器得电状态, TRUE--保持得电,FALSE--断开得电
	enable						:BOOL:=TRUE;//PV禁用条件
	safectrlMode					:BOOL:=FALSE;//eManualCtrMode or eAutoCtrMode
	setPressure					:REAL:=0;// 设置压力值
	configPressure				:REAL:=0;// 配置校准压力
	PressureOffset				:REAL:=1.0;// 压力值偏差
	PositionOffset				:REAL:=1.0;// 位置值偏差
	hmiEN						:BOOL:=TRUE;//HMI 启用条件
	
	errorDelayTime				:TIME:=T#10S;//PV感应器感应超时
	//doneDelayTimeShort		:TIME:=T#100MS;//PV感应到位延时---取消使用
	//doneDelayTimeLong			:TIME:=T#500MS;//无PV感应到位延时---取消使用
	doneDelayTimeShortopen		:TIME:=T#100MS;//PV感应到位延时_打开
	doneDelayTimeShortclose		:TIME:=T#100MS;//PV感应到位延时_关闭
	doneDelayTimeLongopen		:TIME:=T#500MS;//无PV感应到位延时_打开
	doneDelayTimeLongclose		:TIME:=T#500MS;//无PV感应到位延时_关闭
	errorID						:UDINT:=0;//PV错误报警分配的起始ID
	nameTXT						:STRING(255):='';//PV名字
	
	openAprSw					:BOOL:=FALSE;//PV打开感应器信号,需要链接到实际的IO点
	closeAprSw					:BOOL:=FALSE;// PV关闭感应器信号,需要链接到实际的IO点
	enableopenAprSw				:BOOL:=TRUE;//启用打开感应器,针对只有一个传感器的PV
	enablecloseAprSw			:BOOL:=TRUE;// 启用关闭感应器,针对只有一个传感器的PV
	noteWTXT_open				:WSTRING(255):="";//PV打开动作NoteTXT 中文
	noteWTXT_close				:WSTRING(255):="";//PV关闭动作NoteTXT 中文
	configMode					:INT:=0;// 配置模式，不能循环读取数据(0:非Config;1:ZERO;2:PRESSURE ALIGNMENT)
	pvCloseCommunication		:BOOL;// PVClose
	pvOpenCommunication			:BOOL;// PVOpen
	pvPosOrPreCommunication		:BOOL;// PV Pos:=false;Pressure:True;
END_VAR
VAR_OUTPUT
	openRelay				:BOOL:=FALSE;//PV打开执行继电器,需要链接到实际的IO点
	closeRelay				:BOOL:=FALSE;//PV关闭执行继电器,需要链接到实际的IO点
	modeRelay				:BOOL:=FALSE;// PV模式执行继电器,需要链接到实际的IO点
	note_open				:BOOL:=FALSE;// 操作提示：true 打开、打开执行无法下发
	note_close				:BOOL:=FALSE;// 操作提示：true 关闭、关闭执行无法下发
	note_mode				:BOOL:=FALSE;// 操作提示：true Mode切换执行无法下发
	note_config				:BOOL:=FALSE;// 操作提示：true config切换执行无法下发
	busy					:BOOL;//PV动作Busy状态
	done					:BOOL;//PV动作Done状态
	opendone				:BOOL;//PV动作打开完成
	closedone				:BOOL;//PV动作关闭完成
	readdone				:BOOL;// PV读取完成
	modechangedone			:BOOL;// PV模式切换完成
	configdone				:BOOL;// PV配置设置完成
	error					:BOOL;//PV动作error状态
	errID					:UDINT;//PV动作errID
	errTXT					:STRING(255):='';//PV动作errTXT
	errWTXT					:WSTRING(255):="";//PV动作errTXT 中文
	
	serialError				:BOOL:=FALSE;
	contrlmodeRead			:PVControlMOD:=PVControl_Default;// 串口读取回来的控制模式；或者IO都会的串口控制模式
	actPressure				:REAL:=0;// 实际读取的压力值
	actPos					:REAL:=0;// 实际读取的位置值
	openISO					:BOOL;// 开阀
END_VAR
	
VAR		
	serialErrorTimes		:INT:=0;
	readAndWriteLock:BOOL;
	firstPower				:BOOL:=TRUE;
	firstPowerTON			:TON;
	openErrorDelayTon		:Ton;
	openDoneDelayTon		:Ton;
	closeErrorDelayTon		:Ton;
	closeDoneDelayTon		:Ton;
	
	modeErrorDelayTon		:Ton;
	modeDoneDelayTon		:Ton;
	
	openTrigRAlc			:R_Trig;//上升沿触发
	
	openTrigR1				:R_Trig;//上升沿触发
	openTrigF1				:F_Trig;//上升沿触发
	closeTrigR1				:R_Trig;//上升沿触发
	closeTrigF1				:F_Trig;//上升沿触发
	resetTrigR1				:R_Trig;//上升沿触发
	modeTrigR1				:R_Trig;//上升沿触发
	modeTrigF1				:F_Trig;//上升沿触发
	stopTrigR1				:R_Trig;//上升沿触发
	powerTrigR1				:R_Trig;//上升沿触发
	
	setRtrig				:R_Trig;//上升沿触发
	clearRtrig				:R_Trig;//上升沿触发
	configRtrig				:R_Trig;//上升沿触发
	
	openStep				:UINT:=0;
	closeStep				:UINT:=0;
	modeStep				:UINT:=0;
	errorStep				:UINT:=0;
	readStep				:UINT:=0;
	configStep				:UINT:=0;
	
	notBusyMonitorDelayTon:TON;//动作不切换时，延迟检测
	notBusyMonitorDelayTime:TIME:=T#2S;//动作不切换延迟检测时间
	noteTON_P:tON;            // 操作提示标志位延时继电器
	noteTON_N:tON;            // 操作提示标志位延时继电器
	noteRTrig_P:R_TRIG;       // 操作提示
	noteRTrig_N:R_TRIG;       // 操作提示
	opencheckDelayTime	:TON; // 输出到输入检测时间
	openRelayRecTime	:TON; // 输出维持时间
	opencheckDelayTimeS	:TIME; // 输出到输入检测时间
	opencheckRtrig:R_TRIG;     // 输出到输入检测
	closecheckDelayTime	:TON; // 输出到输入检测时间
	closeRelayRecTime	:TON; // 输出维持时间
	closecheckDelayTimeS	:TIME; // 输出到输入检测时间
	closecheckRtrig:R_TRIG;     // 输出到输入检测
	
	oldsetPressure					:REAL:=0;// 压力设置记忆值
	setvalChange					:R_TRIG;// 设置参数变化
	hmiflagReset					:TON;
	readTon1:TON;
	readTon2:TON;
	readTon3:TON;
	configTon1:TON;
	configTon2:TON;
	extRealayRtrig:R_TRIG;
	retRealayRtrig:R_TRIG;
	extRealayRtrig1:R_TRIG;
	retRealayRtrig1:R_TRIG;
	modeRealayRtrig:R_TRIG;
	modeFaleRealayRtrig:R_TRIG;
END_VAR

Init_ACT();
Error_ACT();
open_ACT();
close_ACT();
ModeChange_ACT();
Reset_ACT();
Error_ACT();
SafeMonitor_ACT();
Read_ACT();
ConfigMode_ACT();

(*
触发伸出动作，成功触发返回TRUE，触发失败返回FALSE
*)
METHOD Act_ChangePos : BOOL
VAR_INPUT
END_VAR
IF enable AND modeCondition THEN// AND NOT busy
	HMIItf.mode:=FALSE;
	Act_ChangePos:=mode:=TRUE;
ELSE
	Act_ChangePos:=FALSE;
END_IF
END_METHOD

(*
触发伸出动作，成功触发返回TRUE，触发失败返回FALSE
*)
METHOD Act_ChangePre : BOOL
VAR_INPUT
	setpoint:REAL;
END_VAR
IF enable AND modeCondition THEN// AND NOT busy
	HMIItf.setPressure:=setpoint;
	setPressure:=setPressure;
	HMIItf.mode:=TRUE;
	Act_ChangePre:=mode:=TRUE;
ELSE
	Act_ChangePre:=FALSE;
END_IF
END_METHOD

METHOD Act_Clear : BOOL
VAR_INPUT
END_VAR
setPressure:=0.0;
HMIItf.setPressure:=0.0;
HMIItf.clearflag:=TRUE;
mode:=TRUE;
END_METHOD

(*
触发伸出动作，成功触发返回TRUE，触发失败返回FALSE
*)
METHOD Act_Config : BOOL
VAR_INPUT
END_VAR
IF enable AND configCondition THEN// AND NOT busy
	Act_Config:=config:=TRUE;
ELSE
	Act_Config:=FALSE;
END_IF
END_METHOD

(*
触发伸出动作，成功触发返回TRUE，触发失败返回FALSE
*)
METHOD Act_Open : BOOL
VAR_INPUT
END_VAR
IF enable AND openCondition THEN// AND NOT busy
	Act_Open:=open:=TRUE;
ELSE
	Act_Open:=FALSE;
END_IF
END_METHOD

(*
触发复位报警动作，成功触发返回TRUE，触发失败返回FALSE
*)
METHOD Act_Reset : BOOL
VAR_INPUT
END_VAR
Act_Reset:=reset:=TRUE;
END_METHOD

(*
触发缩回动作，成功触发返回TRUE，触发失败返回FALSE
*)
METHOD Act_Retract : BOOL
VAR_INPUT
END_VAR
IF enable AND closeCondition THEN// AND NOT busy
	Act_Retract:=close:=TRUE;
ELSE
	Act_Retract:=FALSE;
END_IF
END_METHOD

METHOD Act_Set : BOOL
VAR_INPUT
END_VAR
setPressure:=HMIItf.setPressure;
HMIItf.setflag:=TRUE;
mode:=TRUE;
END_METHOD

(*
触发停止输出动作，成功触发返回TRUE，触发失败返回FALSE
*)
METHOD Act_Stop : BOOL
VAR_INPUT
END_VAR
Act_Stop:=stop:=TRUE;
END_METHOD

ACTION Close_ACT:
//气缸收回--close 触发
IF close AND NOT closeCondition THEN
	note_close:=TRUE;
	note_open:=FALSE;
	note_mode:=FALSE;
	note_config:=FALSE;
	NoteHMI.showFlag:=TRUE;
	NoteHMI.showText:='';
	HMIItf.close:=FALSE;
	NoteHMI.showText:=CONCAT(NoteHMI.showText,nameTXT);
	NoteHMI.showText:=CONCAT(NoteHMI.showText,' Close Condition Not Satisfied!');
	operatorLog.append(CONCAT(nameTXT,' Not Close Done '));
END_IF
IF close AND enable AND closeCondition AND  NOT readAndWriteLock THEN// AND NOT busy
	busy:=TRUE;
	open:=FALSE;
	opendone:=FALSE;
	closedone:=FALSE;
	mode:=FALSE;
	modechangedone:=FALSE;
	openStep:=0;
	closeStep:=10;
	modeStep:=0;
	note_open:=FALSE;
	note_close:=FALSE;
	note_config:=FALSE;
	HMIItf.open:=FALSE;
	operatorLog.append(CONCAT(nameTXT,' Close Done '));
	//errorStep:=0;
END_IF
close:=FALSE;
CASE closeStep OF
0:
	//ready
	
10:
	closeErrorDelayTon(IN:=FALSE);
	closeDoneDelayTon(IN:=FALSE);
	closeStep:=20;
	openRelay:=FALSE;
	closeRelay:=TRUE;
	openISO:=FALSE;
	modeRelay:=FALSE;
20:
	closeErrorDelayTon(IN:=((NOT closeAprSw)AND enablecloseAprSw),PT:=errorDelayTime);
	IF closeErrorDelayTon.Q THEN
		//done:=FALSE;
		opendone:=FALSE;
		closedone:=FALSE;
		errorStep:=2;
		RETURN;
	END_IF
	IF enablecloseAprSw THEN
		closeDoneDelayTon(IN:=closeAprSw,PT:=doneDelayTimeShortclose);
	ELSE
		closeDoneDelayTon(IN:=NOT enablecloseAprSw,PT:=doneDelayTimeLongclose);
	END_IF
	
	IF closeDoneDelayTon.Q THEN
		IF NOT openAprSw AND closeAprSw THEN
			busy:=FALSE;
			//done:=TRUE;
			opendone:=FALSE;
			closedone:=TRUE;
			errorStep:=0;
			IF NOT power AND NOT (pvType=PVType_VAT) THEN
				openRelay:=FALSE;
				closeRelay:=FALSE;
			END_IF
			IF pvType=PVType_VAT THEN
				closeRelay:=FALSE;
			END_IF
		ELSE
			busy:=FALSE;
			//done:=TRUE;
			opendone:=FALSE;
			closedone:=FALSE;
			errorStep:=2;
		END_IF
	END_IF
END_CASE
END_ACTION

ACTION ConfigMode_ACT:
//PV打开--config 触发
IF config AND (NOT configCondition OR serialError) THEN
	note_mode:=FALSE;
	note_close:=FALSE;
	note_open:=FALSE;
	note_config:=TRUE;
	NoteHMI.showFlag:=TRUE;
	NoteHMI.showText:='';
	NoteHMI.showText:=CONCAT(NoteHMI.showText,nameTXT);
	NoteHMI.showText:=CONCAT(NoteHMI.showText,' Config Condition Not Satisfied!');
END_IF
IF config AND enable AND configCondition AND NOT serialError AND configMode<>0 AND (configStep<10 OR configStep>39) THEN// AND NOT busy
	busy:=TRUE;
	close:=FALSE;
	mode:=FALSE;
	open:=FALSE;
	configdone:=FALSE;
	configStep:=10;
	modeStep:=0;
	note_open:=FALSE;
	note_close:=FALSE;
	note_mode:=FALSE;
	note_config:=FALSE;
	readAndWriteLock:=TRUE;
	configTon1(IN:=FALSE);
	configTon2(IN:=FALSE);
	//errorStep:=0;
END_IF

config:=FALSE;
CASE configStep OF
0:
	//ready
	
10:
	configTon1(IN:=FALSE);
	configTon2(IN:=FALSE);
	IF (configMode=1 )THEN
		configStep:=20;
		PLC_PDV.WriteZero();
	ELSIF (configMode=2) THEN
		configStep:=30;
		PLC_PDV.WritePressureAlignment(configPressure,2);
	ELSE
		configStep:=40;
	END_IF
20:
	IF (NOT serialError) THEN
		// sendControlModel
		configStep:=22;
	ELSE
		errorStep:=5;
		configStep:=50;// 报错
	END_IF
	configTon1(IN:=FALSE);
	configTon2(IN:=FALSE);
22:
	configTon1(IN:= FALSE(*contrlmodeRead=PVControl_Pressure*),PT:=errorDelayTime);
	IF configTon1.Q THEN
		//done:=FALSE;
		configdone:=FALSE;
		errorStep:=5;
		configTon1(IN:=FALSE);
		configTon2(IN:=FALSE);
		configStep:=50;
		RETURN;
	END_IF
	IF enableopenAprSw THEN
		configTon2(IN:=NOT FALSE(*contrlmodeRead=PVControl_Pressure*),PT:=doneDelayTimeShortopen);
	ELSE
		configTon2(IN:=NOT enableopenAprSw,PT:=doneDelayTimeLongopen);
	END_IF
	IF configTon2.Q THEN
		configStep:=24;
		configTon1(IN:=FALSE);
		configTon2(IN:=FALSE);
	END_IF
24:
	IF (NOT serialError) THEN
		// send Pressure
		configStep:=26;
	ELSE
		errorStep:=5;
		configStep:=50;// 报错
	END_IF
26:
	configTon1(IN:=NOT (TRUE),PT:=errorDelayTime);
	IF configTon1.Q THEN
		//done:=FALSE;
		errorStep:=5;
		configTon1(IN:=FALSE);
		configTon2(IN:=FALSE);
		configStep:=50;
		RETURN;
	END_IF
	IF enableopenAprSw THEN
		configTon2(IN:=TRUE,PT:=doneDelayTimeShortopen);
	ELSE
		configTon2(IN:=NOT enableopenAprSw,PT:=doneDelayTimeLongopen);
	END_IF
	
	IF configTon2.Q THEN
		busy:=FALSE;
		//done:=TRUE;
		configdone:=TRUE;
		errorStep:=0;
		configStep:=40;
		configTon1(IN:=FALSE);
		configTon2(IN:=FALSE);
	END_IF
30:
	IF (NOT serialError) THEN
		// sendControlModel
		configStep:=32;
	ELSE
		errorStep:=5;
		configStep:=50;// 报错
	END_IF
	configTon1(IN:=FALSE);
	configTon2(IN:=FALSE);
32:
	configTon1(IN:= FALSE(*contrlmodeRead=PVControl_Pressure*),PT:=errorDelayTime);
	IF configTon1.Q THEN
		//done:=FALSE;
		configdone:=FALSE;
		errorStep:=5;
		configTon1(IN:=FALSE);
		configTon2(IN:=FALSE);
		configStep:=50;
		RETURN;
	END_IF
	IF enableopenAprSw THEN
		configTon2(IN:=NOT FALSE(*contrlmodeRead=PVControl_Pressure*),PT:=doneDelayTimeShortopen);
	ELSE
		configTon2(IN:=NOT enableopenAprSw,PT:=doneDelayTimeLongopen);
	END_IF
	IF configTon2.Q THEN
		configStep:=34;
		configTon1(IN:=FALSE);
		configTon2(IN:=FALSE);
	END_IF
34:
	IF (NOT serialError) THEN
		// send Pressure
		configStep:=26;
	ELSE
		errorStep:=5;
		configStep:=50;// 报错
	END_IF
36:
	configTon1(IN:=NOT (TRUE),PT:=errorDelayTime);
	IF configTon1.Q THEN
		//done:=FALSE;
		errorStep:=5;
		configTon1(IN:=FALSE);
		configTon2(IN:=FALSE);
		configStep:=50;
		RETURN;
	END_IF
	IF enableopenAprSw THEN
		configTon2(IN:=TRUE,PT:=doneDelayTimeShortopen);
	ELSE
		configTon2(IN:=NOT enableopenAprSw,PT:=doneDelayTimeLongopen);
	END_IF
	
	IF configTon2.Q THEN
		busy:=FALSE;
		//done:=TRUE;
		configdone:=TRUE;
		errorStep:=0;
		configStep:=40;
		configTon1(IN:=FALSE);
		configTon2(IN:=FALSE);
	END_IF
40:
	readAndWriteLock:=FALSE;
50:
	readAndWriteLock:=FALSE;
END_CASE
END_ACTION

ACTION Error_ACT:
CASE errorStep OF
	0:
		error:=FALSE;
		errID:=0;
		errTXT:='';
 (*
	1:
		error:=TRUE;
		errID:=errorID+errorStep;
		errTXT:=CONCAT(STR1:=nameTXT,STR2:=' Extend Error!');
		errWTXT:=WCONCAT(STR1:=TO_WSTRING(nameTXT),STR2:=" 伸出(打开)错误");
	2:
		error:=TRUE;
		errID:=errorID+errorStep;
		errTXT:=CONCAT(STR1:=nameTXT,STR2:=' Retract Error!');
		errWTXT:=WCONCAT(STR1:=TO_WSTRING(nameTXT),STR2:=" 缩回(关闭)错误");
		*)
	1..5:
		error:=TRUE;
		errID:=getErrID(errorStep);
		errTXT:=getErrTXT(errorStep);
		errWTXT:=getErrWTXT(errorStep);
END_CASE
END_ACTION

METHOD Get_Done_Ext : BOOL
VAR_INPUT
END_VAR
Get_Done_Ext:=opendone;
END_METHOD

METHOD Get_Done_Mode : BOOL
VAR_INPUT
END_VAR
Get_Done_Mode:=modechangedone;
END_METHOD

METHOD Get_Done_Ret : BOOL
VAR_INPUT
END_VAR
Get_Done_Ret:=closedone;
END_METHOD

METHOD getErrID : UDINT
VAR_INPUT
	errID					:UDINT;//取值范围1~2
END_VAR
VAR
	nErrID					:UDINT;
END_VAR
nErrID:=errorID+errID;

getErrID:=nErrID;
END_METHOD

METHOD getErrTXT : STRING(255)
VAR_INPUT
	errID					:UDINT;//取值范围1~2
END_VAR
VAR
	sErrTXT					:STRING(255);
END_VAR

CASE errID OF
	1:
		sErrTXT:=CONCAT(STR1:=nameTXT,STR2:=' Open Error!');
	2:
		sErrTXT:=CONCAT(STR1:=nameTXT,STR2:=' Close Error!');
	3:
		sErrTXT:=CONCAT(STR1:=nameTXT,STR2:=' PositionControl Error!');
	4:
		sErrTXT:=CONCAT(STR1:=nameTXT,STR2:=' PressureControl Error!');
	5:
		sErrTXT:=CONCAT(STR1:=nameTXT,STR2:=' Communication Error!');
ELSE
	sErrTXT:=CONCAT(STR1:=nameTXT,STR2:='');
END_CASE
getErrTXT:=sErrTXT;
END_METHOD

METHOD getErrWTXT : WSTRING(255)
VAR_INPUT
	errID					:UDINT;//取值范围1~16
END_VAR
VAR
	sErrTXT					:WSTRING(255);
END_VAR

CASE errID OF
	1:
		sErrTXT:=WCONCAT(STR1:=TO_WSTRING(nameTXT),STR2:=" 伸出(打开)错误");
	2:
		sErrTXT:=WCONCAT(STR1:=TO_WSTRING(nameTXT),STR2:=" 缩回(关闭)错误");
	3:
		sErrTXT:=WCONCAT(STR1:=TO_WSTRING(nameTXT),STR2:=" 位置控制出错");
	4:
		sErrTXT:=WCONCAT(STR1:=TO_WSTRING(nameTXT),STR2:=" 压力控制出错");
	5:
		sErrTXT:=WCONCAT(STR1:=TO_WSTRING(nameTXT),STR2:=" 通讯异常");
ELSE
	sErrTXT:=WCONCAT(STR1:=TO_WSTRING(nameTXT),STR2:="");
END_CASE
getErrWTXT:=sErrTXT;
END_METHOD

ACTION Init_ACT:
done:=(opendone OR closedone);
InitHMI_ACT();
manualCtrl_ACT();

IF serialError OR NOT readCondition AND firstPowerTON.Q THEN
	errorStep:=5;
END_IF
IF (NOT (gICP.PDV.HMIItf.mode) AND ABS(gICP.PDV.HMIItf.setPressure - gICP.PDV.HMIItf.actPos)>1) OR 
   ((gICP.PDV.HMIItf.mode) AND ABS(gICP.PDV.HMIItf.setPressure - gICP.PDV.HMIItf.actPressure)>1) THEN
	HMIItf.setPointNotEq:=TRUE;
ELSE
	HMIItf.setPointNotEq:=FALSE;
END_IF

noteTON_P(IN:=note_open,PT:=T#0.1S);
noteRTrig_P(CLK:=noteTON_P.Q);
IF noteRTrig_P.Q THEN
//	gLog_Note.append_EX(noteWTXT_open);
END_IF
noteTON_N(IN:=note_close,PT:=T#0.1S);
noteRTrig_N(CLK:=noteTON_N.Q);
IF noteRTrig_N.Q THEN
//	gLog_Note.append_EX(noteWTXT_close);
END_IF
modeRealayRtrig(CLK:=modeRelay);
IF modeRealayRtrig.Q THEN
	HMIItf.mode:=TRUE;
END_IF
modeFaleRealayRtrig(CLK:=NOT modeRelay);
IF modeFaleRealayRtrig.Q THEN
	HMIItf.mode:=FALSE;
END_IF

extRealayRtrig(CLK:=openRelay);
IF extRealayRtrig.Q THEN
	HMIItf.open:=TRUE;
END_IF
retRealayRtrig(CLK:=NOT openRelay);
IF retRealayRtrig.Q THEN
	HMIItf.open:=FALSE;
END_IF

extRealayRtrig1(CLK:=closeRelay);
IF extRealayRtrig1.Q THEN
	HMIItf.close:=TRUE;
END_IF
retRealayRtrig1(CLK:=NOT closeRelay);
IF retRealayRtrig1.Q THEN
	HMIItf.close:=FALSE;
END_IF

openRelayRecTime(IN:=openRelay AND (openAprSw OR opendone),PT:=T#0.5S);
IF openRelayRecTime.Q THEN
	HMIItf.open:=FALSE;
END_IF
closeRelayRecTime(IN:=closeRelay AND (closeAprSw OR closedone),PT:=T#0.5S);
IF closeRelayRecTime.Q THEN
	HMIItf.close:=FALSE;
END_IF
END_ACTION

ACTION InitHMI_ACT:
HMIItf.openAprSw:=openAprSw;
HMIItf.closeAprSw:=closeAprSw;
HMIItf.enableopen:=enableopenAprSw;
HMIItf.enableclose:=enablecloseAprSw;
HMIItf.HMIEnable:=hmiEN;
HMIItf.enable:=enable;
HMIItf.done:=done;
HMIItf.busy:=busy;
HMIItf.error:=error;
HMIItf.errID:=UDINT_TO_DINT(errID);
HMIItf.errTXT:=errTXT;
HMIItf.openRelay:=openRelay;
HMIItf.closeRelay:=closeRelay;
HMIItf.power:=power;
HMIItf.nameTXT:=nameTXT;
HMIItf.openerror:=error AND errorID=1;
HMIItf.closeerror:=error AND errorID=2;
HMIItf.opencondition:=openCondition;
HMIItf.closecondition:=closeCondition;

HMIItf.actPos:=actPos;
HMIItf.actPressure:=actPressure;

hmiflagReset(IN:=(HMIItf.clearflag OR HMIItf.setflag),PT:=T#0.2S);
IF hmiflagReset.Q THEN
	HMIItf.clearflag:=FALSE;
	HMIItf.setflag:=FALSE;
END_IF
END_ACTION

ACTION ManualCtrl_ACT:
//HMI手动控制
//IF ctrlMode=eManualCtrMode THEN
IF hmiEN THEN
	openTrigRAlc(CLK:=HMIItf.openAndclose);
	IF openTrigRAlc.Q THEN// AND NOT busy
		IF openRelay THEN//如果伸出继电器或伸出传感器亮，则认为已经伸出过
			close:=TRUE;
		END_IF
		IF closeRelay THEN
			open:=TRUE;
		END_IF
		IF NOT openRelay AND NOT closeRelay THEN
			IF openAprSw THEN
				close:=TRUE;
			END_IF
			IF closeAprSw THEN
				open:=TRUE;
			END_IF
		END_IF
	END_IF
	openTrigR1(CLK:=HMIItf.opentemp);
	openTrigF1(CLK:=HMIItf.open);
	IF openTrigR1.Q THEN// AND NOT busy
		IF NOT HMIItf.open THEN
			WarmHMI.showText:='';
			WarmHMI.showFlag:=TRUE;
			WarmHMI.showText:=CONCAT(WarmHMI.showText,'Are you sure you want to Open the');
			WarmHMI.showText:=CONCAT(WarmHMI.showText,nameTXT);
			WarmHMI.showText:=CONCAT(WarmHMI.showText,' ?');
		ELSE
			HMIItf.open:=FALSE;
		END_IF
	END_IF
	IF WarmHMI.bOK AND NOT WarmHMI.showFlag AND FIND(WarmHMI.showText,nameTXT)>0 AND FIND(WarmHMI.showText,'Open')>0 THEN
		IF HMIItf.open THEN
			;
		ELSE
			open:=TRUE;
			operatorLog.append(CONCAT(nameTXT,' Open'));
		END_IF
		HMIItf.open:=NOT HMIItf.open;
		WarmHMI.bOK:=FALSE;
		WarmHMI.showText:='';
	END_IF
	IF WarmHMI.bNO AND NOT WarmHMI.showFlag AND FIND(WarmHMI.showText,nameTXT)>0 AND FIND(WarmHMI.showText,'Open')>0 THEN
		WarmHMI.bNO:=FALSE;
		WarmHMI.showText:='';
	END_IF
	
	IF openTrigF1.Q THEN// AND NOT busy
		openStep:=0;
		openRelay:=FALSE;
	END_IF
	
	closeTrigR1(CLK:=HMIItf.closetemp);
	closeTrigF1(CLK:=HMIItf.close);
	IF closeTrigR1.Q THEN// AND NOT busy
		IF NOT HMIItf.close THEN
			WarmHMI.showText:='';
			WarmHMI.showFlag:=TRUE;
			WarmHMI.showText:=CONCAT(WarmHMI.showText,'Are you sure you want to Close ');
			WarmHMI.showText:=CONCAT(WarmHMI.showText,nameTXT);
			WarmHMI.showText:=CONCAT(WarmHMI.showText,' ?');
		ELSE
			HMIItf.close:=FALSE;
		END_IF
	END_IF
	IF WarmHMI.bOK AND NOT WarmHMI.showFlag AND FIND(WarmHMI.showText,nameTXT)>0 AND FIND(WarmHMI.showText,'Close')>0 THEN
		IF HMIItf.close THEN
			;
		ELSE
			close:=TRUE;
			operatorLog.append(CONCAT(nameTXT,' Close'));
		END_IF
		HMIItf.close:=NOT HMIItf.close;
		WarmHMI.bOK:=FALSE;
		WarmHMI.showText:='';
	END_IF
	IF WarmHMI.bNO AND NOT WarmHMI.showFlag AND FIND(WarmHMI.showText,nameTXT)>0 AND FIND(WarmHMI.showText,'Close')>0 THEN
		WarmHMI.bNO:=FALSE;
		WarmHMI.showText:='';
	END_IF
	
	IF closeTrigF1.Q THEN// AND NOT busy
		closeStep:=0;
		closeRelay:=FALSE;
	END_IF
	
	modeTrigR1(CLK:=HMIItf.modetemp);
	IF modeTrigR1.Q THEN// AND NOT busy
		HMIItf.modetemp:=FALSE;
		WarmHMI.showText:='';
		WarmHMI.showFlag:=TRUE;
		WarmHMI.showText:=CONCAT(WarmHMI.showText,'Are you sure you want to change the ');
		WarmHMI.showText:=CONCAT(WarmHMI.showText,nameTXT);
		WarmHMI.showText:=CONCAT(WarmHMI.showText,'`Mode ?');
	END_IF
	IF WarmHMI.bOK AND NOT WarmHMI.showFlag AND FIND(WarmHMI.showText,nameTXT)>0 AND FIND(WarmHMI.showText,'Mode')>0 THEN
		mode:=TRUE;
		IF (modeCondition AND NOT serialError) THEN
			HMIItf.mode:=NOT HMIItf.mode;
		END_IF
		operatorLog.append(CONCAT(CONCAT(nameTXT,' Mode Change'),BOOL_TO_STRING(HMIItf.mode)));
		WarmHMI.bOK:=FALSE;
		WarmHMI.showText:='';
	END_IF
	IF WarmHMI.bNO AND NOT WarmHMI.showFlag AND FIND(WarmHMI.showText,nameTXT)>0 AND FIND(WarmHMI.showText,'Mode')>0 THEN
		WarmHMI.bNO:=FALSE;
		WarmHMI.showText:='';
	END_IF
	
	setRtrig(CLK:=HMIItf.set);
	IF setRtrig.Q THEN
		HMIItf.set:=FALSE;
		WarmHMI.showText:='';
		WarmHMI.showFlag:=TRUE;
		WarmHMI.showText:=CONCAT(WarmHMI.showText,'Are you sure you want to Set the ');
		WarmHMI.showText:=CONCAT(WarmHMI.showText,nameTXT);
		WarmHMI.showText:=CONCAT(WarmHMI.showText,'`Par?');
	END_IF
	IF WarmHMI.bOK AND NOT WarmHMI.showFlag AND FIND(WarmHMI.showText,nameTXT)>0 AND FIND(WarmHMI.showText,'Set')>0 THEN
		Act_Set();
		operatorLog.append(CONCAT(CONCAT(nameTXT,' SetPar Change'),REAL_TO_STRING(setPressure)));
		WarmHMI.bOK:=FALSE;
		WarmHMI.showText:='';
	END_IF
	IF WarmHMI.bNO AND NOT WarmHMI.showFlag AND FIND(WarmHMI.showText,nameTXT)>0 AND FIND(WarmHMI.showText,'Set')>0 THEN
		WarmHMI.bNO:=FALSE;
		HMIItf.set:=FALSE;
		WarmHMI.showText:='';
	END_IF
	
	
	
	clearRtrig(CLK:=HMIItf.clear);
	IF clearRtrig.Q THEN
		HMIItf.clear:=FALSE;
		WarmHMI.showText:='';
		WarmHMI.showFlag:=TRUE;
		WarmHMI.showText:=CONCAT(WarmHMI.showText,'Are you sure you want to Clear the ');
		WarmHMI.showText:=CONCAT(WarmHMI.showText,nameTXT);
		WarmHMI.showText:=CONCAT(WarmHMI.showText,'`Par?');
	END_IF
	IF WarmHMI.bOK AND NOT WarmHMI.showFlag AND FIND(WarmHMI.showText,nameTXT)>0 AND FIND(WarmHMI.showText,'Clear')>0 THEN
		Act_Clear();
		operatorLog.append(CONCAT(nameTXT,' Clear'));
		WarmHMI.bOK:=FALSE;
		WarmHMI.showText:='';
	END_IF
	IF WarmHMI.bNO AND NOT WarmHMI.showFlag AND FIND(WarmHMI.showText,nameTXT)>0 AND FIND(WarmHMI.showText,'Clear')>0 THEN
		WarmHMI.bNO:=FALSE;
		HMIItf.clear:=FALSE;
		WarmHMI.showText:='';
	END_IF
	
	configRtrig(CLK:=HMIItf.config);
	IF configRtrig.Q THEN
		HMIItf.config:=FALSE;
		WarmHMI.showText:='';
		WarmHMI.showFlag:=TRUE;
		WarmHMI.showText:=CONCAT(WarmHMI.showText,'Are you sure you want to Config the ');
		WarmHMI.showText:=CONCAT(WarmHMI.showText,nameTXT);
		WarmHMI.showText:=CONCAT(WarmHMI.showText,' ?');
	END_IF
	IF WarmHMI.bOK AND NOT WarmHMI.showFlag AND FIND(WarmHMI.showText,nameTXT)>0 AND FIND(WarmHMI.showText,'Config')>0 THEN
		Act_Config();
		WarmHMI.bOK:=FALSE;
		WarmHMI.showText:='';
	END_IF
	IF WarmHMI.bNO AND NOT WarmHMI.showFlag AND FIND(WarmHMI.showText,nameTXT)>0 AND FIND(WarmHMI.showText,'Config')>0 THEN
		WarmHMI.bNO:=FALSE;
		HMIItf.config:=FALSE;
		WarmHMI.showText:='';
	END_IF
	
	resetTrigR1(CLK:=HMIItf.reset);
	IF resetTrigR1.Q THEN// AND NOT busy
		reset:=TRUE;
	END_IF
	
	stopTrigR1(CLK:=HMIItf.stop);
	IF stopTrigR1.Q THEN// AND NOT busy
		stop:=TRUE;
	END_IF
	
	powerTrigR1(CLK:=HMIItf.power);
	IF powerTrigR1.Q THEN// AND NOT busy
		IF power THEN
			power:=FALSE;
		ELSE
			power:=TRUE;
		END_IF
	END_IF
END_IF
END_ACTION

ACTION ModeChange_ACT:
//PV打开--mode 触发
IF mode AND (NOT modeCondition OR serialError)  THEN
	note_mode:=TRUE;
	note_close:=FALSE;
	note_open:=FALSE;
	note_config:=FALSE;
	NoteHMI.showFlag:=TRUE;
	NoteHMI.showText:='';
	NoteHMI.showText:=CONCAT(NoteHMI.showText,nameTXT);
	NoteHMI.showText:=CONCAT(NoteHMI.showText,' Mode Change Condition Not Satisfied!');
	operatorLog.append(CONCAT(nameTXT,' ModeChange Not Done '));
END_IF
IF mode AND enable AND modeCondition AND NOT serialError AND configMode=0 THEN// AND NOT busy
	busy:=TRUE;
	close:=FALSE;
	mode:=FALSE;
	modechangedone:=FALSE;
	modechangedone:=FALSE;
	IF (actPos<1.0 OR closeAprSw) AND safectrlMode AND openRemOK THEN
		modeStep:=5;
		opencondition_INOUT:=TRUE;
	ELSE
		modeStep:=10;
	END_IF
	note_open:=FALSE;
	note_close:=FALSE;
	note_mode:=FALSE;
	note_config:=FALSE;
	readAndWriteLock:=TRUE;
	operatorLog.append(CONCAT(nameTXT,' ModeChange Done '));
	IF (HMIItf.mode) THEN
		controlMode:=PVControl_Pressure;
	ELSE
		controlMode:=PVControl_Default;
	END_IF
	modeErrorDelayTon(IN:=FALSE);
	modeDoneDelayTon(IN:=FALSE);
	//errorStep:=0;
END_IF
setvalChange(CLK:=oldsetPressure<>setPressure);
oldsetPressure:=setPressure;
mode:=FALSE;
CASE modeStep OF
0:
	//ready
5:
	IF NOT opencondition_INOUT THEN
		opencondition_INOUT:=FALSE;
		modeStep:=10;
	END_IF	
10:
	modeErrorDelayTon(IN:=FALSE);
	modeDoneDelayTon(IN:=FALSE);
	IF (controlMode=PVControl_Default )THEN
		modeRelay:=FALSE;
		modeStep:=20;
		PLC_PDV.WritePositionControl(setPressure,0);
		openISO:=FALSE;
	ELSIF (controlMode=PVControl_Pressure) THEN
		openRelay:=FALSE;
		closeRelay:=FALSE;
		modeRelay:=TRUE;
		PLC_PDV.WritePressureControl(setPressure,0);
		openISO:=TRUE;
		modeStep:=30;
	ELSE
		openRelay:=FALSE;
		closeRelay:=FALSE;
		modeStep:=40;
	END_IF
20:
	IF (NOT serialError) THEN
		// sendControlModel
		modeStep:=22;
	ELSE
		errorStep:=3;
		modeStep:=50;// 报错
	END_IF
	modeErrorDelayTon(IN:=FALSE);
	modeDoneDelayTon(IN:=FALSE);
22:
	modeErrorDelayTon(IN:= modeRelay(*contrlmodeRead=PVControl_Pressure*),PT:=errorDelayTime);
	IF modeErrorDelayTon.Q THEN
		//done:=FALSE;
		opendone:=FALSE;
		closedone:=FALSE;
		errorStep:=3;
		modeErrorDelayTon(IN:=FALSE);
		modeDoneDelayTon(IN:=FALSE);
		modeStep:=50;
		RETURN;
	END_IF
	IF enableopenAprSw THEN
		modeDoneDelayTon(IN:=NOT modeRelay(*contrlmodeRead=PVControl_Pressure*),PT:=doneDelayTimeShortopen);
	ELSE
		modeDoneDelayTon(IN:=NOT enableopenAprSw,PT:=doneDelayTimeLongopen);
	END_IF
	IF modeDoneDelayTon.Q THEN
		modeStep:=24;
		modeErrorDelayTon(IN:=FALSE);
		modeDoneDelayTon(IN:=FALSE);
	END_IF
24:
	IF (NOT serialError) THEN
		// send Pressure
		modeStep:=26;
		readAndWriteLock:=FALSE;
	ELSE
		errorStep:=3;
		modeStep:=50;// 报错
	END_IF
26:
	modeErrorDelayTon(IN:=NOT (ABS(setPressure-actPos)<=PositionOffset),PT:=errorDelayTime);
	IF modeErrorDelayTon.Q THEN
		//done:=FALSE;
		opendone:=FALSE;
		closedone:=FALSE;
		modechangedone:=FALSE;
		errorStep:=3;
		modeStep:=50;
		RETURN;
	END_IF
	IF enableopenAprSw THEN
		modeDoneDelayTon(IN:=ABS(setPressure-actPos)<=PositionOffset,PT:=doneDelayTimeShortopen);
	ELSE
		modeDoneDelayTon(IN:=NOT enableopenAprSw,PT:=doneDelayTimeLongopen);
	END_IF
	
	IF modeDoneDelayTon.Q THEN
		busy:=FALSE;
		//done:=TRUE;
		opendone:=FALSE;
		closedone:=FALSE;
		modechangedone:=TRUE;
		errorStep:=0;
		modeStep:=40;
		modeErrorDelayTon(IN:=FALSE);
		modeDoneDelayTon(IN:=FALSE);
	END_IF
30:
	IF (NOT serialError) THEN
		// sendControlModel
		modeStep:=32;
	ELSE
		errorStep:=4;
		modeStep:=50;// 报错
	END_IF
	modeErrorDelayTon(IN:=FALSE);
	modeDoneDelayTon(IN:=FALSE);
32:
	modeErrorDelayTon(IN:=NOT  modeRelay(*contrlmodeRead=PVControl_Pressure*),PT:=errorDelayTime);
	IF modeErrorDelayTon.Q THEN
		//done:=FALSE;
		opendone:=FALSE;
		closedone:=FALSE;
		errorStep:=4;
		modeErrorDelayTon(IN:=FALSE);
		modeDoneDelayTon(IN:=FALSE);
		modeStep:=50;
		RETURN;
	END_IF
	IF enableopenAprSw THEN
		modeDoneDelayTon(IN:=modeRelay(*contrlmodeRead=PVControl_Pressure*),PT:=doneDelayTimeShortopen);
	ELSE
		modeDoneDelayTon(IN:=NOT enableopenAprSw,PT:=doneDelayTimeLongopen);
	END_IF
	IF modeDoneDelayTon.Q THEN
		modeStep:=34;
		modeErrorDelayTon(IN:=FALSE);
		modeDoneDelayTon(IN:=FALSE);
	END_IF
34:
	IF (NOT serialError) THEN
		// send Pressure
		modeStep:=36;
		readAndWriteLock:=FALSE;
	ELSE
		errorStep:=4;
		modeStep:=50;// 报错
	END_IF
36:
	modeErrorDelayTon(IN:=NOT (ABS(setPressure-actPressure)<=PressureOffset),PT:=errorDelayTime);
	IF modeErrorDelayTon.Q THEN
		//done:=FALSE;
		opendone:=FALSE;
		closedone:=FALSE;
		modechangedone:=FALSE;
		errorStep:=4;
		modeStep:=50;
		RETURN;
	END_IF
	IF enableopenAprSw THEN
		modeDoneDelayTon(IN:=ABS(setPressure-actPressure)<=PressureOffset,PT:=doneDelayTimeShortopen);
	ELSE
		modeDoneDelayTon(IN:=NOT enableopenAprSw,PT:=doneDelayTimeLongopen);
	END_IF
	
	IF modeDoneDelayTon.Q THEN
		busy:=FALSE;
		//done:=TRUE;
		opendone:=FALSE;
		closedone:=FALSE;
		modechangedone:=TRUE;
		errorStep:=0;
		modeStep:=40;
		modeErrorDelayTon(IN:=FALSE);
		modeDoneDelayTon(IN:=FALSE);
	END_IF
40:
	readAndWriteLock:=FALSE;
50:
	readAndWriteLock:=FALSE;
END_CASE
END_ACTION

ACTION Open_ACT:
//PV打开--open 触发
IF open AND NOT openCondition THEN
	note_open:=TRUE;
	note_close:=FALSE;
	note_mode:=FALSE;
	note_config:=FALSE;
	NoteHMI.showFlag:=TRUE;
	HMIItf.open:=FALSE;
	NoteHMI.showText:='';
	NoteHMI.showText:=CONCAT(NoteHMI.showText,nameTXT);
	NoteHMI.showText:=CONCAT(NoteHMI.showText,' Open Condition Not Satisfied!');
	operatorLog.append(CONCAT(nameTXT,' Not Open Done'));
END_IF
IF open AND enable AND openCondition AND NOT readAndWriteLock THEN// AND NOT busy
	busy:=TRUE;
	close:=FALSE;
	opendone:=FALSE;
	closedone:=FALSE;
	mode:=FALSE;
	modechangedone:=FALSE;
	IF (actPos<1.0 OR closeAprSw) AND safectrlMode AND NOT openRemOK THEN
		openStep:=5;
		opencondition_INOUT:=TRUE;
	ELSE
		openStep:=10;
	END_IF
	closeStep:=0;
	modeStep:=0;
	HMIItf.close:=FALSE;
	note_open:=FALSE;
	note_close:=FALSE;
	note_mode:=FALSE;
	note_config:=FALSE;
	operatorLog.append(CONCAT(nameTXT,' Open Done'));
	//errorStep:=0;
END_IF
open:=FALSE;
opencheckDelayTime(IN:=openStep>10 AND NOT opencheckRtrig.Q,PT:=T#60S);
opencheckRtrig(CLK:=openAprSw);
IF opencheckRtrig.Q THEN
	opencheckDelayTimeS:=opencheckDelayTime.ET;
END_IF
CASE openStep OF
0:
	//ready
5:
	IF NOT opencondition_INOUT THEN
		opencondition_INOUT:=FALSE;
		openStep:=10;
	END_IF
10:
	openErrorDelayTon(IN:=FALSE);
	openDoneDelayTon(IN:=FALSE);
	IF (controlMode=PVControl_Default )THEN
		openRelay:=TRUE;
		openISO:=FALSE;
		closeRelay:=FALSE;
		openStep:=20;
	ELSIF (controlMode=PVControl_Pressure) THEN
		openRelay:=FALSE;
		closeRelay:=FALSE;
		openStep:=30;
	ELSE
		openRelay:=FALSE;
		closeRelay:=FALSE;
		openStep:=40;
	END_IF
20:// 位置模式
	openErrorDelayTon(IN:=(((NOT openAprSw OR actPos<99.0) AND controlMode=PVControl_Default) AND enableopenAprSw),PT:=errorDelayTime);
	IF openErrorDelayTon.Q THEN
		//done:=FALSE;
		opendone:=FALSE;
		closedone:=FALSE;
		errorStep:=1;
		RETURN;
	END_IF
	IF enableopenAprSw THEN
		openDoneDelayTon(IN:=(openAprSw AND actPos>99.0 AND controlMode=PVControl_Default) OR controlMode<>PVControl_Default,PT:=doneDelayTimeShortopen);
	ELSE
		openDoneDelayTon(IN:=NOT enableopenAprSw,PT:=doneDelayTimeLongopen);
	END_IF
	
	IF openDoneDelayTon.Q THEN
		IF NOT closeAprSw THEN
			busy:=FALSE;
			//done:=TRUE;
			opendone:=TRUE;
			busy:=FALSE;
			closedone:=FALSE;
			errorStep:=0;
			IF NOT power AND NOT (PVType_VAT=PVType_Default) THEN
				openRelay:=FALSE;
				closeRelay:=FALSE;
			END_IF
			openStep:=40;
			openErrorDelayTon(IN:=FALSE);
			openDoneDelayTon(IN:=FALSE);
		ELSE
			busy:=FALSE;
			//done:=TRUE;
			opendone:=FALSE;
			closedone:=FALSE;
			errorStep:=1;
		END_IF
	END_IF
30:
	IF (NOT serialError) THEN
		// sendControlModel
		openStep:=32;
	ELSE
		errorStep:=5;
		openStep:=50;// 报错
	END_IF
32:
	openErrorDelayTon(IN:=NOT (contrlmodeRead=PVControl_Pressure),PT:=errorDelayTime);
	IF openErrorDelayTon.Q THEN
		//done:=FALSE;
		opendone:=FALSE;
		closedone:=FALSE;
		errorStep:=1;
		openErrorDelayTon(IN:=FALSE);
		openDoneDelayTon(IN:=FALSE);
		RETURN;
	END_IF
	IF enableopenAprSw THEN
		openDoneDelayTon(IN:=(contrlmodeRead=PVControl_Pressure),PT:=doneDelayTimeShortopen);
	ELSE
		openDoneDelayTon(IN:=NOT enableopenAprSw,PT:=doneDelayTimeLongopen);
	END_IF
	IF openDoneDelayTon.Q THEN
		openStep:=34;
		openErrorDelayTon(IN:=FALSE);
		openDoneDelayTon(IN:=FALSE);
	END_IF
34:
	IF (NOT serialError) THEN
		// send Pressure
		openStep:=36;
	ELSE
		errorStep:=5;
		openStep:=50;// 报错
	END_IF
36:
	openErrorDelayTon(IN:=NOT (ABS(setPressure-actPressure)<PressureOffset AND actPos>0.01),PT:=errorDelayTime);
	IF openErrorDelayTon.Q THEN
		//done:=FALSE;
		opendone:=FALSE;
		closedone:=FALSE;
		errorStep:=1;
		openStep:=50;// 报错
		RETURN;
	END_IF
	IF enableopenAprSw THEN
		openDoneDelayTon(IN:=ABS(setPressure-actPressure)<PressureOffset AND actPos>0.01,PT:=doneDelayTimeShortopen);
	ELSE
		openDoneDelayTon(IN:=NOT enableopenAprSw,PT:=doneDelayTimeLongopen);
	END_IF
	
	IF openDoneDelayTon.Q THEN
		IF NOT closeAprSw THEN
			busy:=FALSE;
			//done:=TRUE;
			opendone:=TRUE;
			closedone:=FALSE;
			errorStep:=0;
			openStep:=40;
			openErrorDelayTon(IN:=FALSE);
			openDoneDelayTon(IN:=FALSE);
		ELSE
			busy:=FALSE;
			//done:=TRUE;
			opendone:=FALSE;
			closedone:=FALSE;
			errorStep:=1;
			openStep:=50;// 报错
			openErrorDelayTon(IN:=FALSE);
			openDoneDelayTon(IN:=FALSE);
		END_IF
	END_IF
END_CASE
END_ACTION

ACTION Read_ACT:
//气缸收回--read 触发
firstPowerTON(IN:=firstPower,PT:=T#10S);
IF NOT readAndWriteLock AND readStep=0 AND readCondition AND configMode=0 THEN// AND NOT busy
	readdone:=FALSE;
	readStep:=10;
END_IF
CASE readStep OF
0:
	//ready
	readTon1(IN:=FALSE);
	readTon2(IN:=FALSE);
	readTon3(IN:=FALSE);
10:// State
	IF readAndWriteLock THEN
		readStep:=5000;
	ELSE
		PLC_PDV.readStateFlag:=FALSE;
		PLC_PDV.ReadState();
		readStep:=readStep+10;
	END_IF
20:
	IF readAndWriteLock THEN
		readStep:=5000;
	ELSE
		IF PLC_PDV.readStateFlag THEN
			PLC_PDV.readStateFlag:=FALSE;
			// 数据处理
			readTon1(IN:=FALSE);
			readStep:=readStep+10;
			pvCloseCommunication:=PLC_PDV.pvCloseCommunication;
			pvOpenCommunication:=PLC_PDV.pvOpenCommunication;
			pvPosOrPreCommunication:=PLC_PDV.pvPosOrPreCommunication;
			serialErrorTimes:=0;
			serialError:=FALSE;
			RETURN;
		END_IF
		readTon1(IN:=TRUE,PT:=T#500MS);// 超时
		IF readTon1.Q THEN
			readStep:=6000;
			readTon1(IN:=FALSE);
			readTon2(IN:=FALSE);
			serialErrorTimes:=serialErrorTimes+1;
			RETURN;
		END_IF
		;
	END_IF
30:
	readTon3(IN:=TRUE,PT:=T#50MS);
	IF readTon3.Q THEN
		readTon1(IN:=FALSE);
		readTon2(IN:=FALSE);
		readTon3(IN:=FALSE);
		IF serialErrorTimes>10 THEN
			serialErrorTimes:=0;
			serialError:=TRUE;
		END_IF
		readStep:=100;
	END_IF
100:// Internal Pressure
	IF readAndWriteLock THEN
		readStep:=5000;
	ELSE
		PLC_PDV.readPressureFlag:=FALSE;
		PLC_PDV.ReadPressure();
		readStep:=readStep+10;
	END_IF	
110:
	IF readAndWriteLock THEN
		readStep:=5000;
	ELSE
		IF PLC_PDV.readPressureFlag THEN
			PLC_PDV.readPressureFlag:=FALSE;
			// 数据处理
			readTon1(IN:=FALSE);
			readStep:=readStep+10;
			actPressure:=INT_TO_REAL(PLC_PDV.pvReadPre);
			serialErrorTimes:=0;
			serialError:=FALSE;
			RETURN;
		END_IF
		readTon1(IN:=TRUE,PT:=T#500MS);// 超时
		IF readTon1.Q THEN
			readStep:=6000;
			readTon1(IN:=FALSE);
			readTon2(IN:=FALSE);
			serialErrorTimes:=serialErrorTimes+1;
			RETURN;
		END_IF
		;
	END_IF
120:
	readTon3(IN:=TRUE,PT:=T#50MS);
	IF readTon3.Q THEN
		readTon1(IN:=FALSE);
		readTon2(IN:=FALSE);
		readTon3(IN:=FALSE);
		IF serialErrorTimes>10 THEN
			serialErrorTimes:=0;
			serialError:=TRUE;
		END_IF
		readStep:=200;
	END_IF
	
200:// External ReadPosition
	IF readAndWriteLock THEN
		readStep:=5000;
	ELSE
		PLC_PDV.readPostitionFlag:=FALSE;
		PLC_PDV.ReadPosition();
		readStep:=readStep+10;
	END_IF
210:
	IF readAndWriteLock THEN
		readStep:=5000;
	ELSE
		IF PLC_PDV.readPostitionFlag THEN
			PLC_PDV.readPostitionFlag:=FALSE;
			// 数据处理
			readTon1(IN:=FALSE);
			readStep:=readStep+10;
			actPos:=INT_TO_REAL(PLC_PDV.pvReadPos);
			serialErrorTimes:=0;
			serialError:=FALSE;
			RETURN;
		END_IF
		readTon1(IN:=TRUE,PT:=T#500MS);// 超时
		IF readTon1.Q THEN
			readStep:=6000;
			readTon1(IN:=FALSE);
			readTon2(IN:=FALSE);
			serialErrorTimes:=serialErrorTimes+1;
			RETURN;
		END_IF
		;
	END_IF
220:
	readTon3(IN:=TRUE,PT:=T#50MS);
	IF readTon3.Q THEN
		readTon1(IN:=FALSE);
		readTon2(IN:=FALSE);
		readTon3(IN:=FALSE);
		IF serialErrorTimes>10 THEN
			serialErrorTimes:=0;
			serialError:=TRUE;
		END_IF
		readStep:=5000;
	END_IF
5000:
	readdone:=TRUE;
	readStep:=0;
	IF serialErrorTimes>10 THEN
		serialErrorTimes:=0;
		serialError:=TRUE;
	END_IF
6000:
	readdone:=TRUE;
	readStep:=0;
	IF serialErrorTimes>10 THEN
		serialErrorTimes:=0;
		serialError:=TRUE;
	END_IF
END_CASE
END_ACTION

ACTION Reset_ACT:
IF reset THEN
	IF NOT power THEN
		openRelay:=FALSE;
		closeRelay:=FALSE;
	END_IF
	busy:=FALSE;
	//done:=FALSE;
	//opendone:=FALSE;
	//closedone:=FALSE;
	errorStep:=0;
	IF error THEN
		IF opencondition_INOUT THEN
			openStep:=0;
			opencondition_INOUT:=FALSE;
		END_IF
	END_IF
	note_open:=FALSE;
	note_close:=FALSE;
	reset:=FALSE;
END_IF

IF stop AND error THEN
	stop:=FALSE;
	openRelay:=FALSE;
	closeRelay:=FALSE;
	// 控制模式是否需要清除归零
	note_open:=FALSE;
	note_close:=FALSE;
	//无自锁检测说法，直接停
//	openStep:=0;
//	closeStep:=0;
END_IF
END_ACTION

ACTION SafeMonitor_ACT:
notBusyMonitorDelayTon(IN:=NOT busy,PT:=notBusyMonitorDelayTime);
IF real_TimeMonitor THEN
	IF notBusyMonitorDelayTon.Q AND contrlmodeRead=PVControl_Default THEN
		//伸出实时检测
		IF (enableopenAprSw AND NOT openAprSw) AND openRelay THEN
			errorStep:=1;
		END_IF
	
